// NeuroPLC — Auto-generated IEC 61131-3 SCL
// Graph: kan | Target: S71200Backend
// Work memory: 75KB | LUT points: 15
// Nodes: 11 | Ops: {'matmul': 3, 'standard_act': 2, 'bspline_lut': 2, 'add': 2, 'softmax': 1, 'argmax': 1}


DATA_BLOCK "NeuroPLC_Weights"
{ S7_Optimized_Access := 'FALSE' }
VERSION : 0.1
NON_RETAIN
   STRUCT

   // BsplineLUT 'l0_bspline': grid(15 pts) + table(16×28×15)
   w0 : ARRAY[0..14] OF REAL :=
[-3.0000000, -2.5714286, -2.1428571, -1.7142857, -1.2857143, -0.8571429, -0.4285714, 0.0
    0.4285714, 0.8571429, 1.2857143, 1.7142857, 2.1428571, 2.5714286, 3.0000000];
   w1 : ARRAY[0..6719] OF REAL :=
[-0.0064954, -0.0050089, -0.0033770, -0.0016958, -0.0000479, 0.0014853, 0.0028220, 0.0038805
    0.0045846, 0.0048793, 0.0047147, 0.0040414, 0.0028094, 0.0009775, -0.0013529, -0.0130491
    -0.0087791, -0.0036095, 0.0020238, 0.0073062, 0.0114015, 0.0134733, 0.0126853, 0.0084933
    0.0015210, -0.0073160, -0.0171017, -0.0269205, -0.0358740, -0.0433676, -0.0119517, -0.0074362
    -0.0021026, 0.0035783, 0.0087589, 0.0125698, 0.0141418, 0.0126054, 0.0074143, -0.0006864
    -0.0106286, -0.0213443, -0.0317654, -0.0408502, -0.0480129, -0.0055758, -0.0085337, -0.0109214
    -0.0123673, -0.0124829, -0.0108790, -0.0071661, -0.0009551, 0.0079073, 0.0186290, 0.0301819
    0.0415377, 0.0516683, 0.0595823, 0.0649290, 0.0033017, -0.0018919, -0.0086076, -0.0158108
    -0.0218283, -0.0249507, -0.0234683, -0.0156713, -0.0006975, 0.0189270, 0.0398287, 0.0586340
    0.0719694, 0.0766010, 0.0717208, -0.0145982, -0.0132009, -0.0118636, -0.0105667, -0.0090013
    -0.0068415, -0.0037615, 0.0005645, 0.0063401, 0.0132795, 0.0209750, 0.0290186, 0.0370023
    0.0445224, 0.0512483, 0.0005540, 0.0050713, 0.0109763, 0.0176704, 0.0237023, 0.0275720
    0.0277792, 0.0228238, 0.0116819, -0.0047655, -0.0251609, -0.0481471, -0.0723664, -0.0964808
    -0.1194836, -0.0025839, -0.0029541, -0.0026654, -0.0016455, 0.0000022, 0.0021641, 0.0047267
    0.0075767, 0.0104673, 0.0126194, 0.0131209, 0.0110596, 0.0055231, -0.0043401, -0.0183258
    -0.0085053, -0.0092509, -0.0093235, -0.0085654, -0.0068801, -0.0041745, -0.0003556, 0.0046696
    0.0108291, 0.0173902, 0.0234552, 0.0281264, 0.0305059, 0.0297509, 0.0259743, -0.0022033
    -0.0008497, 0.0003257, 0.0012372, 0.0018995, 0.0023330, 0.0025581, 0.0025952, 0.0024489
    0.0020599, 0.0013534, 0.0002540, -0.0013131, -0.0034131, -0.0059392, 0.0570825, 0.0523418
    0.0441618, 0.0326389, 0.0183960, 0.0020866, -0.0156358, -0.0341180, -0.0527775, -0.0713162
    -0.0895071, -0.1071230, -0.1239369, -0.1396837, -0.1534356, -0.0017276, 0.0135975, 0.0262822
    0.0349414, 0.0388797, 0.0374410, 0.0299697, 0.0158097, -0.0051883, -0.0311484, -0.0596881
    -0.0884251, -0.1149769, -0.1370229, -0.1533197, 0.0417430, 0.0132695, -0.0117596, -0.0313531
    -0.0452569, -0.0533167, -0.0553782, -0.0512872, -0.0412373, -0.0268139, -0.0099504, 0.0074197
    0.0233633, 0.0360149, 0.0446960, 0.0591801, 0.0506987, 0.0420201, 0.0335674, 0.0251025
    0.0163496, 0.0070328, -0.0031239, -0.0142303, -0.0257320, -0.0369083, -0.0470387, -0.0554027
    -0.0613104, -0.0646050, 0.0380552, 0.0305894, 0.0203781, 0.0079362, -0.0053995, -0.0182449
    -0.0292158, -0.0369281, -0.0402260, -0.0388668, -0.0328362, -0.0221198, -0.0067033, 0.0133397
    0.0364058, -0.0794777, -0.0800806, -0.0797186, -0.0782858, -0.0752684, -0.0701291, -0.0623306
    -0.0513354, -0.0369371, -0.0202517, -0.0027264, 0.0141921, 0.0290567, 0.0404752, 0.0480044
    -0.1608721, -0.1544616, -0.1423316, -0.1249372, -0.1034885, -0.0792385, -0.0534405, -0.0273477
    -0.0021188, 0.0214652, 0.0427176, 0.0609519, 0.0754814, 0.0856493, 0.0913159, 0.0539866
    0.0477996, 0.0377296, 0.0240342, 0.0077611, -0.0099963, -0.0281447, -0.0455906, -0.0613476
    -0.0748558, -0.0856624, -0.0933141, -0.0973580, -0.0973787, -0.0936133, 0.0534758, 0.0429142
    0.0305485, 0.0172136, 0.0040506, -0.0077813, -0.0171231, -0.0228160, -0.0239895, -0.0209286
    -0.0142067, -0.0043974, 0.0079257, 0.0221621, 0.0372402, 0.1102775, 0.1072526, 0.1021108
    0.0946131, 0.0838261, 0.0687763, 0.0484902, 0.0219946, -0.0109618, -0.0477404, -0.0849806
    -0.1193216, -0.1474027, -0.1660319, -0.1749534, -0.0983728, -0.0679108, -0.0389890, -0.0138788
    0.0064673, 0.0211730, 0.0293616, 0.0301567, 0.0231331, 0.0096706, -0.0083994, -0.0292456
    -0.0510370, -0.0719598, -0.0905098, -0.1422940, -0.1310264, -0.1130547, -0.0893668, -0.0624104
    -0.0347168, -0.0088174, 0.0127565, 0.0280181, 0.0371596, 0.0409174, 0.0400284, 0.0352292
    0.0272730, 0.0171998, -0.1772897, -0.1588601, -0.1331439, -0.1010212, -0.0656541, -0.0303357
    0.0016410, 0.0269829, 0.0431205, 0.0503784, 0.0498048, 0.0424480, 0.0293561, 0.0116197
    -0.0089316, -0.0924975, -0.0685450, -0.0453334, -0.0240949, -0.0058931, 0.0082184, 0.0171858
    0.0199555, 0.0158568, 0.0057512, -0.0091168, -0.0275026, -0.0481617, -0.0698275, -0.0908472
    -0.0919868, -0.0763941, -0.0599793, -0.0435190, -0.0277131, -0.0132577, -0.0008484, 0.0088188
    0.0152255, 0.0185620, 0.0191960, 0.0174953, 0.0138274, 0.0085720, 0.0023131, -0.1375341
    -0.1143461, -0.0884176, -0.0609049, -0.0337633, -0.0089942, 0.0114009, 0.0254207, 0.0315517
    0.0302322, 0.0223883, 0.0089463, -0.0091677, -0.0309746, -0.0545734, -0.0019394, 0.0037786
    0.0098244, 0.0154883, 0.0197382, 0.0215240, 0.0197951, 0.0135014, 0.0019694, -0.0139657
    -0.0330918, -0.0541969, -0.0760687, -0.0974818, -0.1169787, -0.1755243, -0.1531998, -0.1266178
    -0.0966809, -0.0651036, -0.0336468, -0.0040715, 0.0218613, 0.0427145, 0.0583474, 0.0689429
    0.0746840, 0.0757539, 0.0723667, 0.0652806, -0.0696934, -0.0602897, -0.0487975, -0.0357825
    -0.0218667, -0.0076757, 0.0061653, 0.0190307, 0.0302458, 0.0389377, 0.0441842, 0.0450629
    0.0406516, 0.0301205, 0.0142489, -0.0597138, -0.0559139, -0.0494283, -0.0404261, -0.0294536
    -0.0170791, -0.0038708, 0.0096030, 0.0226738, 0.0342706, 0.0432220, 0.0483568, 0.0485035
    0.0425778, 0.0310126, -0.0605716, -0.0569390, -0.0505317, -0.0415093, -0.0304389, -0.0179108
    -0.0045154, 0.0091569, 0.0224174, 0.0341838, 0.0432753, 0.0485114, 0.0487112, 0.0427819
    0.0311602, -0.0516885, -0.0380645, -0.0247713, -0.0127368, -0.0022508, 0.0064337, 0.0130636
    0.0173857, 0.0192439, 0.0188696, 0.0165911, 0.0127368, 0.0076349, 0.0016172, -0.0049279
    -0.0562407, -0.0516357, -0.0434013, -0.0321080, -0.0191705, -0.0060523, 0.0057832, 0.0148725
    0.0201440, 0.0220925, 0.0216043, 0.0195661, 0.0168642, 0.0143631, 0.0125459, -0.0215669
    -0.0173831, -0.0123562, -0.0067542, -0.0009397, 0.0047195, 0.0098553, 0.0140999, 0.0171329
    0.0188250, 0.0190945, 0.0178597, 0.0150389, 0.0105708, 0.0047481, -0.0566579, -0.0562306
    -0.0548574, -0.0523959, -0.0483627, -0.0422548, -0.0335695, -0.0218037, -0.0067783, 0.0103907
    0.0282635, 0.0454004, 0.0603615, 0.0717702, 0.0793456, -0.0520496, -0.0423928, -0.0325770
    -0.0232095, -0.0144005, -0.0062322, 0.0012138, 0.0078554, 0.0136411, 0.0186406, 0.0229540
    0.0266813, 0.0299225, 0.0327781, 0.0353559, -0.0642884, -0.0507025, -0.0367111, -0.0231770
    -0.0104224, 0.0012616, 0.0115839, 0.0202534, 0.0269396, 0.0311546, 0.0323713, 0.0300626
    0.0237013, 0.0128268, -0.0018600, -0.0367120, -0.0243320, -0.0127388, -0.0027711, 0.0054115
    0.0116887, 0.0159399, 0.0180448, 0.0179132, 0.0155768, 0.0110978, 0.0045382, -0.0040400
    -0.0145496, -0.0264691, -0.1216510, -0.1105591, -0.0941895, -0.0733171, -0.0496326, -0.0248794
    -0.0008011, 0.0208591, 0.0387466, 0.0530622, 0.0643957, 0.0733367, 0.0804749, 0.0863647
    0.0909459, -0.0027857, -0.0084430, -0.0145285, -0.0204270, -0.0250927, -0.0274549, -0.0264427
    -0.0209856, -0.0104698, 0.0038897, 0.0204213, 0.0374528, 0.0533125, 0.0663794, 0.0759185
    0.0129611, 0.0254017, 0.0356314, 0.0425417, 0.0455004, 0.0439032, 0.0371453, 0.0246222
    0.0061932, -0.0164266, -0.0410586, -0.0655236, -0.0876430, -0.1053033, -0.1175339, -0.0247634
    -0.0279660, -0.0288906, -0.0272312, -0.0232430, -0.0172134, -0.0094298, -0.0001796, 0.0101667
    0.0209071, 0.0312566, 0.0404302, 0.0476427, 0.0521333, 0.0535592, -0.1293642, -0.1193707
    -0.1032642, -0.0817289, -0.0568370, -0.0307407, -0.0055918, 0.0164574, 0.0336519, 0.0458234
    0.0532008, 0.0560128, 0.0544880, 0.0488898, 0.0400817, 0.0759348, 0.0751573, 0.0733678
    0.0703268, 0.0651676, 0.0569878, 0.0448845, 0.0279552, 0.0058174, -0.0198302, -0.0467688
    -0.0727795, -0.0956434, -0.1132157, -0.1246400, 0.0752203, 0.0702935, 0.0637723, 0.0558556
    0.0465078, 0.0356797, 0.0233220, 0.0093856, -0.0060020, -0.0220067, -0.0376174, -0.0518232
    -0.0636131, -0.0720135, -0.0767006, -0.1173986, -0.1049409, -0.0871985, -0.0650950, -0.0405694
    -0.0156189, 0.0077592, 0.0275678, 0.0422579, 0.0520735, 0.0577069, 0.0598503, 0.0591959
    0.0564281, 0.0520940, -0.1212512, -0.1127163, -0.0993807, -0.0818294, -0.0613756, -0.0393746
    -0.0171817, 0.0038479, 0.0225291, 0.0383576, 0.0509995, 0.0601208, 0.0653873, 0.0665038
    0.0638503, -0.1056125, -0.1031581, -0.0990820, -0.0934024, -0.0856393, -0.0752838, -0.0618274
    -0.0447613, -0.0239545, -0.0007861, 0.0229867, 0.0456071, 0.0653182, 0.0804434, 0.0907060
    0.0487952, 0.0374115, 0.0242019, 0.0102135, -0.0029327, -0.0135830, -0.0200835, -0.0207803
    -0.0146193, -0.0029447, 0.0122998, 0.0291703, 0.0457231, 0.0600643, 0.0711699, 0.0646500
    0.0612506, 0.0529924, 0.0403731, 0.0250127, 0.0085953, -0.0071945, -0.0206726, -0.0303979
    -0.0359026, -0.0369623, -0.0333526, -0.0248490, -0.0113090, 0.0059815, 0.0825636, 0.0740969
    0.0609729, 0.0435120, 0.0233914, 0.0023661, -0.0178087, -0.0353779, -0.0489058, -0.0582347
    -0.0635260, -0.0649415, -0.0626425, -0.0568210, -0.0481953, 0.0733571, 0.0654811, 0.0543846
    0.0404885, 0.0252671, 0.0102550, -0.0030131, -0.0130025, -0.0185798, -0.0202170, -0.0187870
    -0.0151632, -0.0102187, -0.0048108, 0.0004789, 0.0597846, 0.0506018, 0.0387739, 0.0250072
    0.0108969, -0.0019105, -0.0117689, -0.0170321, -0.0165256, -0.0109636, -0.0015320, 0.0105832
    0.0241959, 0.0381237, 0.0512467, 0.0794086, 0.0712941, 0.0590351, 0.0430848, 0.0252648
    0.0074750, -0.0083842, -0.0204127, -0.0271671, -0.0290304, -0.0268422, -0.0214424, -0.0136706
    -0.0043701, 0.0055541, -0.0189963, -0.0221225, -0.0233823, -0.0223317, -0.0191588, -0.0140878
    -0.0073429, 0.0008515, 0.0102233, 0.0203094, 0.0305988, 0.0405802, 0.0497428, 0.0575804
    0.0636721, 0.0415532, 0.0397687, 0.0360804, 0.0306095, 0.0239207, 0.0166041, 0.0092500
    0.0024485, -0.0033091, -0.0079269, -0.0114082, -0.0137560, -0.0149734, -0.0150717, -0.0142024
    -0.1213656, -0.1098515, -0.0929578, -0.0714629, -0.0470719, -0.0215433, 0.0033646, 0.0258933
    0.0444176, 0.0578437, 0.0652110, 0.0655589, 0.0579266, 0.0414757, 0.0174933, -0.1205001
    -0.1097379, -0.0932614, -0.0718080, -0.0471914, -0.0212873, 0.0040288, 0.0268811, 0.0455475
    0.0589196, 0.0660424, 0.0659608, 0.0577200, 0.0404886, 0.0155879, -0.1202567, -0.1093710
    -0.0927757, -0.0712194, -0.0465306, -0.0206000, 0.0046820, 0.0274247, 0.0458997, 0.0590270
    0.0658889, 0.0655675, 0.0571451, 0.0398251, 0.0149239, -0.0930097, -0.0831860, -0.0703592
    -0.0552040, -0.0386853, -0.0217846, -0.0054833, 0.0092369, 0.0215748, 0.0314497, 0.0389614
    0.0442093, 0.0472932, 0.0483230, 0.0475881, -0.1132518, -0.1079017, -0.0976854, -0.0829627
    -0.0649007, -0.0447129, -0.0236130, -0.0028146, 0.0165543, 0.0337069, 0.0479419, 0.0585582
    0.0648543, 0.0661755, 0.0626742, -0.0815116, -0.0730840, -0.0626569, -0.0507423, -0.0377882
    -0.0242390, -0.0105393, 0.0028667, 0.0155580, 0.0272082, 0.0375145, 0.0461741, 0.0528842
    0.0573621, 0.0596777, -0.1008868, -0.0948195, -0.0856380, -0.0736700, -0.0594149, -0.0433822
    -0.0260816, -0.0080224, 0.0102401, 0.0279682, 0.0443783, 0.0586871, 0.0701108, 0.0779097
    0.0821002, -0.0928198, -0.0838908, -0.0722195, -0.0583813, -0.0431031, -0.0271209, -0.0111703
    0.0040129, 0.0177917, 0.0299241, 0.0402667, 0.0486763, 0.0550096, 0.0591411, 0.0612585
    -0.1192025, -0.1073053, -0.0904778, -0.0695176, -0.0459871, -0.0214926, 0.0023598, 0.0239637
    0.0418163, 0.0548291, 0.0620169, 0.0623945, 0.0549769, 0.0389000, 0.0154086, -0.0679830
    -0.0513064, -0.0341468, -0.0177486, -0.0029976, 0.0092411, 0.0181021, 0.0227202, 0.0224813
    0.0177747, 0.0092409, -0.0024797, -0.0167467, -0.0329079, -0.0501083, -0.1202152, -0.1092289
    -0.0926936, -0.0714178, -0.0472899, -0.0222603, 0.0017207, 0.0227027, 0.0392099, 0.0516649
    0.0609646, 0.0680063, 0.0736871, 0.0788536, 0.0834750, -0.0320415, -0.0206113, -0.0114709
    -0.0052510, -0.0012089, 0.0014771, 0.0036287, 0.0060675, 0.0094544, 0.0138069, 0.0189818
    0.0248359, 0.0312257, 0.0379923, 0.0447006, 0.0660699, 0.0630954, 0.0595871, 0.0554868
    0.0500426, 0.0424626, 0.0319549, 0.0177277, -0.0005979, -0.0217477, -0.0440348, -0.0657718
    -0.0852719, -0.1008953, -0.1118326, 0.0328585, 0.0217698, 0.0119434, 0.0043030, -0.0008504
    -0.0032515, -0.0026349, 0.0012646, 0.0083698, 0.0172324, 0.0260619, 0.0330673, 0.0364579
    0.0345348, 0.0271977, -0.1172725, -0.1090614, -0.0961407, -0.0789738, -0.0588449, -0.0370850
    -0.0150253, 0.0060030, 0.0248866, 0.0413825, 0.0554658, 0.0671113, 0.0762938, 0.0829856
    0.0871120, 0.0788702, 0.0767232, 0.0737037, 0.0696657, 0.0637522, 0.0550650, 0.0427063
    0.0257779, 0.0038922, -0.0212971, -0.0476260, -0.0729304, -0.0950462, -0.1118830, -0.1226330
    0.0424648, 0.0355723, 0.0284807, 0.0217434, 0.0156830, 0.0106090, 0.0068309, 0.0046579
    0.0042683, 0.0053151, 0.0073201, 0.0098052, 0.0122921, 0.0143158, 0.0156396, -0.1141555
    -0.1016998, -0.0839089, -0.0618142, -0.0376349, -0.0136582, 0.0078285, 0.0245378, 0.0347400
    0.0389358, 0.0381833, 0.0335407, 0.0260662, 0.0168141, 0.0067709, -0.1213959, -0.1175703
    -0.1110765, -0.1020365, -0.0903403, -0.0758647, -0.0584862, -0.0380815, -0.0148199, 0.0099586
    0.0346216, 0.0575365, 0.0770708, 0.0916617, 0.1009580, -0.0431900, -0.0438981, -0.0437770
    -0.0425988, -0.0398651, -0.0350619, -0.0276752, -0.0171910, -0.0033860, 0.0128013, 0.0301419
    0.0474065, 0.0633661, 0.0768385, 0.0874577, 0.0019430, -0.0087142, -0.0163489, -0.0201806
    -0.0205530, -0.0178746, -0.0125535, -0.0049983, 0.0043352, 0.0147992, 0.0256987, 0.0363382
    0.0460225, 0.0540709, 0.0600565, 0.0039094, 0.0201128, 0.0296586, 0.0319383, 0.0287980
    0.0222250, 0.0142065, 0.0067297, 0.0014772, -0.0010882, -0.0008081, 0.0024758, 0.0089216
    0.0186273, 0.0306427, 0.0763165, 0.0725086, 0.0658738, 0.0564109, 0.0447281, 0.0314686
    0.0172757, 0.0027923, -0.0114108, -0.0250536, -0.0379287, -0.0498286, -0.0605459, -0.0698632
    -0.0773902, 0.0831831, 0.0795113, 0.0726465, 0.0625293, 0.0497289, 0.0348502, 0.0184983
    0.0012784, -0.0162054, -0.0333528, -0.0495646, -0.0642413, -0.0767837, -0.0866050, -0.0933383
    0.0471839, 0.0355534, 0.0222393, 0.0082356, -0.0048220, -0.0152611, -0.0214091, -0.0215935
    -0.0147504, -0.0022505, 0.0139268, 0.0318021, 0.0493961, 0.0647776, 0.0768565, 0.0713515
    0.0666394, 0.0594218, 0.0498125, 0.0385150, 0.0262667, 0.0138048, 0.0018668, -0.0089300
    -0.0184476, -0.0266677, -0.0335724, -0.0391433, -0.0433604, -0.0461668, -0.0771443, -0.0710582
    -0.0617116, -0.0493296, -0.0350074, -0.0198900, -0.0051224, 0.0081503, 0.0190202, 0.0275273
    0.0339489, 0.0385621, 0.0416443, 0.0434640, 0.0441410, -0.0979009, -0.0862316, -0.0711662
    -0.0531324, -0.0335126, -0.0137440, 0.0047361, 0.0204905, 0.0323993, 0.0406117, 0.0455938
    0.0478122, 0.0477332, 0.0458205, 0.0424930, 0.0944311, 0.0863878, 0.0740996, 0.0580816
    0.0395634, 0.0198158, 0.0001096, -0.0182844, -0.0341089, -0.0461598, -0.0532464, -0.0541781
    -0.0477642, -0.0329385, -0.0108025, 0.0939177, 0.0870638, 0.0758494, 0.0606509, 0.0425458
    0.0226521, 0.0020875, -0.0180299, -0.0364904, -0.0517164, -0.0620384, -0.0657868, -0.0612920
    -0.0470345, -0.0241054, 0.0934611, 0.0864068, 0.0749925, 0.0596162, 0.0413892, 0.0214640
    0.0009928, -0.0188720, -0.0369049, -0.0515887, -0.0613327, -0.0645465, -0.0596398, -0.0451677
    -0.0222238, 0.0570179, 0.0537455, 0.0489764, 0.0428718, 0.0355747, 0.0272273, 0.0179716
    0.0079496, -0.0025564, -0.0127039, -0.0215103, -0.0279928, -0.0311689, -0.0301138, -0.0249110
    0.0460533, 0.0528679, 0.0571354, 0.0582993, 0.0560601, 0.0501329, 0.0402327, 0.0260748
    0.0077565, -0.0130960, -0.0344739, -0.0543687, -0.0707718, -0.0817546, -0.0867803, 0.0621695
    0.0584621, 0.0535885, 0.0476425, 0.0404141, 0.0316758, 0.0212000, 0.0087594, -0.0055780
    -0.0205620, -0.0346468, -0.0462869, -0.0539364, -0.0561275, -0.0527471, 0.0701987, 0.0696979
    0.0675516, 0.0635566, 0.0572396, 0.0481121, 0.0356854, 0.0194707, -0.0006887, -0.0236225
    -0.0478285, -0.0718046, -0.0940486, -0.1131139, -0.1285232, 0.0605322, 0.0579419, 0.0539998
    0.0487406, 0.0420048, 0.0336216, 0.0234203, 0.0112302, -0.0029310, -0.0182922, -0.0338936
    -0.0487758, -0.0619792, -0.0725872, -0.0804313, 0.0925140, 0.0843020, 0.0722705, 0.0569652
    0.0395218, 0.0211099, 0.0028993, -0.0139404, -0.0282564, -0.0389630, -0.0449914, -0.0452728
    -0.0387385, -0.0244341, -0.0033994, 0.0693646, 0.0566685, 0.0426540, 0.0284249, 0.0152002
    0.0042055, -0.0033339, -0.0061924, -0.0035427, 0.0038494, 0.0148200, 0.0282050, 0.0428405
    0.0575849, 0.0716867, 0.0069745, 0.0062506, 0.0064994, 0.0078262, 0.0099654, 0.0126300
    0.0155331, 0.0183876, 0.0208833, 0.0226164, 0.0231599, 0.0220866, 0.0189695, 0.0134287
    0.0059034, 0.0326397, 0.0199406, 0.0098152, 0.0032476, 0.0000372, -0.0000846, 0.0026136
    0.0078633, 0.0152792, 0.0240088, 0.0330832, 0.0415332, 0.0483899, 0.0527224, 0.0542676
    0.0053282, 0.0129482, 0.0183251, 0.0210448, 0.0216541, 0.0207547, 0.0189484, 0.0168371
    0.0149329, 0.0133894, 0.0122708, 0.0116410, 0.0115643, 0.0120930, 0.0130789, -0.0381531
    -0.0262031, -0.0143655, -0.0034747, 0.0060392, 0.0137694, 0.0193090, 0.0222511, 0.0224485
    0.0207927, 0.0184346, 0.0165254, 0.0162159, 0.0186006, 0.0237847, 0.0409369, 0.0423051
    0.0424320, 0.0410951, 0.0380820, 0.0331813, 0.0261813, 0.0168703, 0.0052438, -0.0078751
    -0.0214561, -0.0344691, -0.0458837, -0.0547040, -0.0605266, 0.0091396, 0.0119548, 0.0140948
    0.0154324, 0.0161025, 0.0162550, 0.0160399, 0.0156069, 0.0150929, 0.0145815, 0.0141431
    0.0138481, 0.0137671, 0.0139622, 0.0143534, 0.0721669, 0.0742674, 0.0740355, 0.0712051
    0.0656274, 0.0571602, 0.0456614, 0.0309891, 0.0132578, -0.0063905, -0.0265570, -0.0458430
    -0.0628498, -0.0762186, -0.0852870, -0.0089771, -0.0124859, -0.0142004, -0.0137117, -0.0110339
    -0.0062053, 0.0007355, 0.0097502, 0.0206647, 0.0327626, 0.0451921, 0.0571012, 0.0676379
    0.0759713, 0.0816357, 0.0681135, 0.0717669, 0.0731730, 0.0718734, 0.0674359, 0.0594302
    0.0474258, 0.0309923, 0.0101209, -0.0135104, -0.0378020, -0.0606542, -0.0799673, -0.0937302
    -0.1014727, 0.0066072, 0.0131599, 0.0193168, 0.0245588, 0.0284010, 0.0303603, 0.0299538
    0.0266985, 0.0203090, 0.0112903, 0.0003451, -0.0118241, -0.0245147, -0.0370358, -0.0489014
    -0.1054841, -0.0859640, -0.0655508, -0.0454745, -0.0263027, -0.0085651, 0.0072089, 0.0204895
    0.0308788, 0.0385047, 0.0436267, 0.0465041, 0.0473965, 0.0465646, 0.0442899, 0.0230305
    0.0095048, 0.0011872, -0.0014041, 0.0002786, 0.0046702, 0.0102053, 0.0153185, 0.0186618
    0.0197552, 0.0183360, 0.0141414, 0.0069087, -0.0035626, -0.0163892, -0.1229653, -0.1097450
    -0.0931571, -0.0735213, -0.0519821, -0.0297309, -0.0079594, 0.0121409, 0.0296408, 0.0446615
    0.0575863, 0.0687990, 0.0786830, 0.0875849, 0.0952085, -0.1548740, -0.1414460, -0.1227592
    -0.0991485, -0.0722224, -0.0436623, -0.0151498, 0.0116337, 0.0353166, 0.0557683, 0.0731680
    0.0876950, 0.0995286, 0.1088290, 0.1154228, -0.1086425, -0.0899576, -0.0683922, -0.0451821
    -0.0221343, -0.0010883, 0.0161161, 0.0276392, 0.0321437, 0.0303009, 0.0232844, 0.0122680
    -0.0015748, -0.0170612, -0.0328486, -0.1558141, -0.1408449, -0.1207802, -0.0960685, -0.0684270
    -0.0396461, -0.0115157, 0.0141738, 0.0359979, 0.0539937, 0.0685638, 0.0801109, 0.0890376
    0.0957244, 0.1001640, -0.0616598, -0.0524274, -0.0414076, -0.0290780, -0.0160703, -0.0030250
    0.0094170, 0.0206151, 0.0300767, 0.0379012, 0.0443362, 0.0496289, 0.0540270, 0.0577579
    0.0607039, 0.0925081, 0.0809107, 0.0674662, 0.0525844, 0.0372056, 0.0223005, 0.0088397
    -0.0022058, -0.0100878, -0.0149464, -0.0171444, -0.0170443, -0.0150086, -0.0114080, -0.0067522
    -0.1215551, -0.1098357, -0.0927275, -0.0710164, -0.0464081, -0.0206612, 0.0044657, 0.0272140
    0.0459589, 0.0596108, 0.0672138, 0.0678120, 0.0604495, 0.0442920, 0.0206181, -0.1208857
    -0.1095647, -0.0924934, -0.0704504, -0.0453027, -0.0189797, 0.0065890, 0.0294740, 0.0479249
    0.0609077, 0.0675675, 0.0670493, 0.0584981, 0.0411776, 0.0164150, -0.1205362, -0.1090672
    -0.0918623, -0.0697141, -0.0445053, -0.0181810, 0.0073136, 0.0300334, 0.0482226, 0.0608837
    0.0672086, 0.0663892, 0.0576175, 0.0402015, 0.0154702, -0.0941092, -0.0845557, -0.0718859
    -0.0567428, -0.0400791, -0.0228652, -0.0060714, 0.0093319, 0.0225441, 0.0334438, 0.0420794
    0.0484995, 0.0527524, 0.0548977, 0.0551881, -0.1170871, -0.1116646, -0.1013879, -0.0865732
    -0.0683226, -0.0477831, -0.0261021, -0.0044266, 0.0161521, 0.0347672, 0.0506076, 0.0628627
    0.0707213, 0.0734210, 0.0710410, -0.0823846, -0.0739108, -0.0634201, -0.0514188, -0.0383376
    -0.0246032, -0.0106423, 0.0031187, 0.0162708, 0.0284763, 0.0394149, 0.0487667, 0.0562115
    0.0614492, 0.0645269, -0.0991079, -0.0922577, -0.0822467, -0.0694684, -0.0545329, -0.0380632
    -0.0206821, -0.0030123, 0.0143144, 0.0306304, 0.0452592, 0.0575243, 0.0667490, 0.0722997
    0.0742855, -0.0928475, -0.0838840, -0.0721083, -0.0580921, -0.0425772, -0.0263157, -0.0100593
    0.0054401, 0.0195247, 0.0319125, 0.0424159, 0.0508468, 0.0570176, 0.0607599, 0.0622474
    -0.1203630, -0.1085233, -0.0916387, -0.0704921, -0.0466520, -0.0217322, 0.0026534, 0.0248913
    0.0434635, 0.0572356, 0.0651691, 0.0662254, 0.0593662, 0.0436765, 0.0203970, -0.0680496
    -0.0515522, -0.0344431, -0.0179460, -0.0029658, 0.0096107, 0.0188968, 0.0240060, 0.0243005
    0.0201390, 0.0121289, 0.0008778, -0.0130066, -0.0289036, -0.0459612, -0.1138717, -0.1025615
    -0.0859516, -0.0648777, -0.0412208, -0.0169221, 0.0060774, 0.0258366, 0.0408898, 0.0516737
    0.0591004, 0.0640818, 0.0675302, 0.0703143, 0.0725504, -0.0350313, -0.0229405, -0.0128055
    -0.0053238, 0.0000572, 0.0039619, 0.0070147, 0.0098400, 0.0129439, 0.0163589, 0.0199993
    0.0237792, 0.0276129, 0.0314070, 0.0349383, 0.0761654, 0.0712323, 0.0657907, 0.0599320
    0.0529649, 0.0441535, 0.0327617, 0.0180532, -0.0003224, -0.0211741, -0.0429252, -0.0639990
    -0.0828190, -0.0978532, -0.1083473, 0.0390785, 0.0275469, 0.0171428, 0.0088180, 0.0028944
    -0.0003426, -0.0006074, 0.0023855, 0.0085804, 0.0165564, 0.0245516, 0.0308039, 0.0335512
    0.0311235, 0.0234511, -0.1124076, -0.1048866, -0.0926845, -0.0762174, -0.0567367, -0.0355421
    -0.0139333, 0.0067902, 0.0255361, 0.0420414, 0.0562504, 0.0681074, 0.0775567, 0.0845398
    0.0889506, 0.0777938, 0.0761875, 0.0736788, 0.0700997, 0.0646103, 0.0563323, 0.0443873
    0.0278971, 0.0064857, -0.0182131, -0.0440628, -0.0689272, -0.0906700, -0.1072281, -0.1178123
    0.0306264, 0.0248821, 0.0192516, 0.0142293, 0.0100919, 0.0071031, 0.0055270, 0.0056275
    0.0075227, 0.0107481, 0.0146931, 0.0187473, 0.0223004, 0.0247633, 0.0259229, -0.1100040
    -0.0974996, -0.0798112, -0.0579656, -0.0341471, -0.0106065, 0.0104052, 0.0266372, 0.0363968
    0.0402233, 0.0392138, 0.0344657, 0.0270764, 0.0181347, 0.0085847, -0.1101300, -0.1074096
    -0.1023327, -0.0949400, -0.0850188, -0.0723417, -0.0566813, -0.0378103, -0.0158138, 0.0079732
    0.0319032, 0.0543286, 0.0736020, 0.0881442, 0.0975696, -0.0224207, -0.0236837, -0.0245226
    -0.0247033, -0.0237885, -0.0213294, -0.0168772, -0.0099832, -0.0004217, 0.0111389, 0.0238074
    0.0366923, 0.0489020, 0.0595761, 0.0683924, -0.0233470, -0.0315586, -0.0356521, -0.0350509
    -0.0305355, -0.0229643, -0.0131955, -0.0020877, 0.0095558, 0.0211516, 0.0321712, 0.0420859
    0.0503673, 0.0565039, 0.0602835, -0.0084433, 0.0087051, 0.0199937, 0.0247043, 0.0244047
    0.0207943, 0.0155723, 0.0104381, 0.0068485, 0.0052909, 0.0060104, 0.0092522, 0.0152612
    0.0242227, 0.0352821, 0.0585067, 0.0569909, 0.0533496, 0.0474729, 0.0396850, 0.0303350
    0.0197723, 0.0083458, -0.0035997, -0.0157382, -0.0277479, -0.0393072, -0.0500946, -0.0597806
    -0.0678997, 0.0763782, 0.0748911, 0.0701328, 0.0619394, 0.0508106, 0.0372841, 0.0218974
    0.0051883, -0.0122721, -0.0297793, -0.0465951, -0.0619815, -0.0752003, -0.0855319, -0.0925743
    0.0374300, 0.0266855, 0.0146888, 0.0023938, -0.0087210, -0.0171474, -0.0213768, -0.0199010
    -0.0117905, 0.0015674, 0.0182065, 0.0361603, 0.0534627, 0.0681992, 0.0793608, 0.0584625
    0.0558492, 0.0511390, 0.0443516, 0.0359860, 0.0265690, 0.0166272, 0.0066872, -0.0027968
    -0.0116610, -0.0198142, -0.0271652, -0.0336226, -0.0390905, -0.0433884, -0.0890283, -0.0810995
    -0.0695774, -0.0548310, -0.0381366, -0.0208221, -0.0042159, 0.0103538, 0.0218367, 0.0302932
    0.0360615, 0.0394797, 0.0408862, 0.0406171, 0.0389746, -0.1011540, -0.0898113, -0.0746058
    -0.0559599, -0.0353910, -0.0144791, 0.0051956, 0.0220529, 0.0348570, 0.0437498, 0.0492174
    0.0517461, 0.0518220, 0.0499288, 0.0465025, -0.1150191, -0.1040288, -0.0878393, -0.0671941
    -0.0437533, -0.0192299, 0.0046633, 0.0262135, 0.0438444, 0.0565260, 0.0633650, 0.0634681
    0.0559420, 0.0400093, 0.0169120, -0.1136940, -0.1035435, -0.0878935, -0.0674332, -0.0439016
    -0.0190980, 0.0051784, 0.0271281, 0.0450974, 0.0580147, 0.0649535, 0.0649878, 0.0571912
    0.0407560, 0.0169362, -0.1135426, -0.1032815, -0.0875194, -0.0669554, -0.0433427, -0.0184950
    0.0057740, 0.0276506, 0.0454741, 0.0581963, 0.0649221, 0.0647562, 0.0568036, 0.0402859
    0.0164578, -0.0887678, -0.0792654, -0.0668474, -0.0521640, -0.0361579, -0.0197886, -0.0040159
    0.0102007, 0.0220788, 0.0315445, 0.0387009, 0.0436513, 0.0464988, 0.0473565, 0.0465069
    -0.1083338, -0.1028552, -0.0927300, -0.0783368, -0.0608156, -0.0413501, -0.0211241, -0.0013213
    0.0169684, 0.0330303, 0.0462434, 0.0559867, 0.0616393, 0.0626229, 0.0591023, -0.0775478
    -0.0695332, -0.0595474, -0.0480733, -0.0355557, -0.0224369, -0.0091594, 0.0038346, 0.0161274
    0.0274012, 0.0373626, 0.0457186, 0.0521761, 0.0564617, 0.0586449, -0.0962942, -0.0905587
    -0.0818326, -0.0704136, -0.0567581, -0.0413319, -0.0246004, -0.0070292, 0.0108738, 0.0284328
    0.0449295, 0.0596457, 0.0718633, 0.0809003, 0.0867065, -0.0886533, -0.0800715, -0.0688260
    -0.0554658, -0.0406965, -0.0252327, -0.0097892, 0.0049194, 0.0182786, 0.0300741, 0.0401918
    0.0485174, 0.0549369, 0.0593518, 0.0619392, -0.1129163, -0.1014855, -0.0853049, -0.0651442
    -0.0425303, -0.0190337, 0.0037750, 0.0243255, 0.0411600, 0.0532720, 0.0597679, 0.0597540
    0.0523366, 0.0367359, 0.0141528, -0.0644862, -0.0485097, -0.0320092, -0.0161761, -0.0018866
    0.0100011, 0.0186287, 0.0231381, 0.0229192, 0.0183537, 0.0100715, -0.0012977, -0.0151239
    -0.0307667, -0.0473992, -0.1192922, -0.1084692, -0.0920533, -0.0708351, -0.0467016, -0.0216032
    0.0025099, 0.0236875, 0.0404533, 0.0532275, 0.0629040, 0.0703769, 0.0765402, 0.0822354
    0.0873918, -0.0294734, -0.0189659, -0.0106106, -0.0049696, -0.0013039, 0.0012005, 0.0033573
    0.0059804, 0.0097195, 0.0145674, 0.0203531, 0.0269052, 0.0340527, 0.0416067, 0.0490741
    0.0650349, 0.0627376, 0.0597952, 0.0561095, 0.0509495, 0.0435475, 0.0331361, 0.0189477
    0.0006264, -0.0205367, -0.0428393, -0.0645787, -0.0840523, -0.0996066, -0.1104411, 0.0299549
    0.0195369, 0.0103629, 0.0033123, -0.0013214, -0.0032781, -0.0022979, 0.0018792, 0.0091779
    0.0181812, 0.0271367, 0.0342920, 0.0378948, 0.0362825, 0.0293554, -0.1136357, -0.1055042
    -0.0927660, -0.0758810, -0.0561190, -0.0347965, -0.0132299, 0.0072643, 0.0255859, 0.0414988
    0.0549833, 0.0660195, 0.0745876, 0.0806665, 0.0842130, 0.0796799, 0.0776106, 0.0746405
    0.0706247, 0.0647179, 0.0560345, 0.0436891, 0.0267961, 0.0049771, -0.0201172, -0.0463292
    -0.0715011, -0.0934753, -0.1101679, -0.1207850, 0.0471702, 0.0401892, 0.0328941, 0.0258325
    0.0193094, 0.0136164, 0.0090447, 0.0058856, 0.0043172, 0.0040642, 0.0047380, 0.0059499
    0.0073114, 0.0084452, 0.0091719, -0.1143654, -0.1021862, -0.0845330, -0.0624114, -0.0380585
    -0.0137824, 0.0081091, 0.0253079, 0.0360626, 0.0408471, 0.0406915, 0.0366261, 0.0296812
    0.0208831, 0.0111921, -0.1183035, -0.1140783, -0.1073372, -0.0982326, -0.0866561, -0.0724844
    -0.0555943, -0.0358624, -0.0134468, 0.0103689, 0.0340196, 0.0559402, 0.0745657, 0.0883988
    0.0971212, -0.0449943, -0.0453366, -0.0448266, -0.0432475, -0.0400870, -0.0348164, -0.0269064
    -0.0158281, -0.0013547, 0.0155321, 0.0335481, 0.0514091, 0.0678313, 0.0815803, 0.0922910
    0.0065674, -0.0063583, -0.0157020, -0.0205504, -0.0213812, -0.0187517, -0.0132195, -0.0053419
    0.0043035, 0.0150584, 0.0262445, 0.0371835, 0.0471970, 0.0556191, 0.0620026, 0.0105306
    0.0255404, 0.0339575, 0.0352378, 0.0312270, 0.0239082, 0.0152645, 0.0072789, 0.0016253
    -0.0012590, -0.0012459, 0.0017927, 0.0079849, 0.0174008, 0.0291002, 0.0858274, 0.0804212
    0.0722181, 0.0612891, 0.0482883, 0.0339036, 0.0188229, 0.0037340, -0.0107619, -0.0244099
    -0.0370420, -0.0484899, -0.0585854, -0.0671524, -0.0738745, 0.0880742, 0.0826101, 0.0743533
    0.0633208, 0.0500298, 0.0350263, 0.0188560, 0.0020649, -0.0148010, -0.0311950, -0.0465703
    -0.0603800, -0.0720773, -0.0811279, -0.0872167, 0.0517958, 0.0393813, 0.0254100, 0.0109012
    -0.0025541, -0.0133320, -0.0198087, -0.0203604, -0.0139593, -0.0019614, 0.0136811, 0.0310161
    0.0480916, 0.0630035, 0.0746856, 0.0802013, 0.0737863, 0.0650000, 0.0540316, 0.0416047
    0.0284741, 0.0153943, 0.0031199, -0.0077261, -0.0170466, -0.0248760, -0.0312489, -0.0361996
    -0.0397611, -0.0419380, -0.0813725, -0.0748128, -0.0649224, -0.0519620, -0.0370499, -0.0213537
    -0.0060409, 0.0077209, 0.0190091, 0.0278806, 0.0346374, 0.0395811, 0.0430137, 0.0452262
    0.0463194, -0.0887788, -0.0781593, -0.0643381, -0.0476983, -0.0295392, -0.0112124, 0.0059304
    0.0205375, 0.0315560, 0.0391289, 0.0436976, 0.0457040, 0.0455896, 0.0437931, 0.0406991
    -0.0681019, -0.0558745, -0.0441106, -0.0335166, -0.0238243, -0.0147096, -0.0058486, 0.0030829
    0.0123038, 0.0216121, 0.0307007, 0.0392626, 0.0469907, 0.0535900, 0.0589749, -0.0745009
    -0.0610971, -0.0466884, -0.0322327, -0.0184111, -0.0058885, 0.0046702, 0.0125999, 0.0175007
    0.0200328, 0.0211215, 0.0216920, 0.0226695, 0.0249387, 0.0286753, -0.0721163, -0.0584018
    -0.0438990, -0.0295951, -0.0161466, -0.0041911, 0.0056340, 0.0126911, 0.0166200, 0.0181703
    0.0183687, 0.0182420, 0.0188171, 0.0210736, 0.0251719, -0.0926290, -0.0828816, -0.0707450
    -0.0568312, -0.0417447, -0.0260898, -0.0104708, 0.0045080, 0.0182859, 0.0304758, 0.0407343
    0.0487180, 0.0540833, 0.0565155, 0.0561972, -0.0907978, -0.0859772, -0.0774038, -0.0652007
    -0.0502352, -0.0334171, -0.0156562, 0.0021376, 0.0190963, 0.0345190, 0.0477468, 0.0581205
    0.0649812, 0.0677005, 0.0661841, -0.0552471, -0.0429697, -0.0313496, -0.0211351, -0.0121846
    -0.0043050, 0.0026963, 0.0090124, 0.0147835, 0.0199395, 0.0243578, 0.0279157, 0.0304905
    0.0319690, 0.0324008, -0.0518637, -0.0356115, -0.0191431, -0.0037401, 0.0095546, 0.0197123
    0.0257038, 0.0265003, 0.0214690, 0.0115618, -0.0018731, -0.0174878, -0.0339341, -0.0498954
    -0.0646034, -0.0750934, -0.0627938, -0.0492242, -0.0351928, -0.0212449, -0.0079108, 0.0042793
    0.0147952, 0.0231211, 0.0287994, 0.0313867, 0.0304399, 0.0255157, 0.0162241, 0.0031023
    -0.0756219, -0.0651536, -0.0545072, -0.0442427, -0.0341002, -0.0237729, -0.0129537, -0.0013358
    0.0112176, 0.0241618, 0.0367822, 0.0483640, 0.0581923, 0.0655877, 0.0704843, -0.0199903
    -0.0168361, -0.0138871, -0.0112165, -0.0084661, -0.0052529, -0.0011937, 0.0040943, 0.0108419
    0.0186709, 0.0270508, 0.0354510, 0.0433412, 0.0502094, 0.0558684, -0.0951167, -0.0843383
    -0.0687285, -0.0492257, -0.0279636, -0.0071445, 0.0110293, 0.0243556, 0.0311273, 0.0316189
    0.0266003, 0.0168414, 0.0031120, -0.0137778, -0.0323163, -0.0324504, -0.0335040, -0.0301457
    -0.0224050, -0.0118296, -0.0000543, 0.0112860, 0.0205565, 0.0263758, 0.0283759, 0.0264421
    0.0204599, 0.0103147, -0.0040378, -0.0214172, 0.0946146, 0.0857759, 0.0748829, 0.0623615
    0.0483462, 0.0329548, 0.0163048, -0.0014860, -0.0201712, -0.0389892, -0.0570498, -0.0734627
    -0.0873376, -0.0978102, -0.1044702, 0.0510492, 0.0419094, 0.0334937, 0.0264414, 0.0206468
    0.0159612, 0.0122362, 0.0093230, 0.0070724, 0.0053317, 0.0039475, 0.0027665, 0.0016353
    0.0004161, -0.0007572, -0.1006878, -0.0916718, -0.0785101, -0.0617960, -0.0429373, -0.0233887
    -0.0046048, 0.0119598, 0.0251807, 0.0352542, 0.0427072, 0.0480662, 0.0518579, 0.0545862
    0.0563552, 0.0503459, 0.0532122, 0.0547124, 0.0544169, 0.0517122, 0.0459743, 0.0365792
    0.0229029, 0.0047388, -0.0164501, -0.0387834, -0.0603808, -0.0793618, -0.0939094, -0.1033076
    -0.0408732, -0.0338215, -0.0260637, -0.0179739, -0.0096838, -0.0013109, 0.0070272, 0.0152130
    0.0230338, 0.0298967, 0.0351137, 0.0379967, 0.0378577, 0.0340710, 0.0270941, -0.1021982
    -0.0930440, -0.0790383, -0.0608542, -0.0401324, -0.0185691, 0.0021393, 0.0202965, 0.0346070
    0.0453794, 0.0533228, 0.0591466, 0.0635600, 0.0672356, 0.0702077, 0.0692438, 0.0678171
    0.0636722, 0.0568775, 0.0478867, 0.0371755, 0.0252196, 0.0124947, -0.0004698, -0.0129301
    -0.0240889, -0.0331487, -0.0393122, -0.0418328, -0.0408491, 0.0921181, 0.0916542, 0.0900433
    0.0870802, 0.0819053, 0.0736216, 0.0613323, 0.0441403, 0.0216763, -0.0043176, -0.0315718
    -0.0578167, -0.0807825, -0.0983015, -0.1099787, -0.1119333, -0.1013238, -0.0848411, -0.0631974
    -0.0384422, -0.0127021, 0.0118965, 0.0332272, 0.0495246, 0.0604681, 0.0660983, 0.0664555
    0.0615804, 0.0515728, 0.0375695, -0.0730997, -0.0675506, -0.0572406, -0.0428076, -0.0259146
    -0.0082835, 0.0083640, 0.0223060, 0.0322131, 0.0383257, 0.0412767, 0.0416989, 0.0402252
    0.0374778, 0.0338920, -0.1076191, -0.0973288, -0.0817078, -0.0611327, -0.0375210, -0.0128788
    0.0107878, 0.0314728, 0.0476305, 0.0595576, 0.0680112, 0.0737484, 0.0775264, 0.0800688
    0.0815150, -0.0741057, -0.0625820, -0.0490312, -0.0339187, -0.0182590, -0.0030981, 0.0105180
    0.0215433, 0.0292440, 0.0341347, 0.0370423, 0.0387934, 0.0402149, 0.0420890, 0.0444250
    -0.0928475, -0.0842471, -0.0718093, -0.0558799, -0.0377289, -0.0186795, -0.0000546, 0.0168227
    0.0308220, 0.0415834, 0.0489398, 0.0527240, 0.0527690, 0.0489501, 0.0418835, -0.1074911
    -0.0975065, -0.0823477, -0.0623628, -0.0394076, -0.0154245, 0.0076440, 0.0278558, 0.0436803
    0.0552340, 0.0630454, 0.0676432, 0.0695555, 0.0693021, 0.0672456, -0.1037187, -0.0934545
    -0.0781682, -0.0583332, -0.0359152, -0.0129661, 0.0084626, 0.0263191, 0.0389774, 0.0465126
    0.0494256, 0.0482171, 0.0433880, 0.0354613, 0.0253502, -0.0266544, -0.0336035, -0.0358269
    -0.0331325, -0.0266085, -0.0174167, -0.0067191, 0.0043226, 0.0147216, 0.0241911, 0.0326196
    0.0398955, 0.0459071, 0.0505421, 0.0536739, -0.0570067, -0.0510674, -0.0426060, -0.0319958
    -0.0200086, -0.0074390, 0.0049183, 0.0162687, 0.0258464, 0.0330016, 0.0371130, 0.0375598
    0.0337208, 0.0250448, 0.0121974, -0.0520371, -0.0486492, -0.0428014, -0.0346550, -0.0247561
    -0.0136728, -0.0019731, 0.0097748, 0.0209302, 0.0305615, 0.0376646, 0.0412354, 0.0402695
    0.0338457, 0.0224826, -0.0525712, -0.0493106, -0.0435266, -0.0353693, -0.0253905, -0.0141650
    -0.0022675, 0.0097271, 0.0211668, 0.0310908, 0.0384612, 0.0422399, 0.0413890, 0.0349552
    0.0234615, -0.0436548, -0.0344229, -0.0244913, -0.0145098, -0.0049960, 0.0035400, 0.0105880
    0.0156380, 0.0183099, 0.0187436, 0.0172091, 0.0139763, 0.0093153, 0.0035013, -0.0030965
    -0.0556900, -0.0499911, -0.0410367, -0.0294721, -0.0165975, -0.0037504, 0.0077314, 0.0165105
    0.0216022, 0.0234336, 0.0227849, 0.0204365, 0.0171684, 0.0137455, 0.0106627, -0.0259741
    -0.0219326, -0.0168972, -0.0111316, -0.0050199, 0.0010473, 0.0066791, 0.0114847, 0.0151220
    0.0174439, 0.0183521, 0.0177483, 0.0155340, 0.0116302, 0.0062922, -0.0511092, -0.0508130
    -0.0497722, -0.0478703, -0.0446635, -0.0396890, -0.0324842, -0.0225864, -0.0097885, 0.0050931
    0.0209868, 0.0368205, 0.0515223, 0.0640591, 0.0740691, -0.0455572, -0.0389769, -0.0315846
    -0.0238023, -0.0159021, -0.0081477, -0.0008025, 0.0058698, 0.0116732, 0.0166817, 0.0210367
    0.0248796, 0.0283520, 0.0315941, 0.0347292, -0.0521327, -0.0440120, -0.0343157, -0.0235823
    -0.0124407, -0.0015250, 0.0085306, 0.0170920, 0.0235774, 0.0276143, 0.0288828, 0.0270626
    0.0218338, 0.0129269, 0.0009554, -0.0296755, -0.0206468, -0.0117076, -0.0034971, 0.0036499
    0.0094163, 0.0134849, 0.0155384, 0.0153486, 0.0130434, 0.0088394, 0.0029535, -0.0043976
    -0.0129850, -0.0223708, -0.1298479, -0.1198579, -0.1037237, -0.0821519, -0.0570350, -0.0303334
    -0.0040077, 0.0199815, 0.0400947, 0.0564755, 0.0696887, 0.0802990, 0.0888711, 0.0959336
    0.1013906, -0.0123170, -0.0173108, -0.0223907, -0.0269699, -0.0300543, -0.0306267, -0.0276697
    -0.0201659, -0.0075500, 0.0089352, 0.0275948, 0.0467340, 0.0646579, 0.0797176, 0.0910631
    0.0070675, 0.0216721, 0.0336126, 0.0416478, 0.0452635, 0.0439874, 0.0373472, 0.0248705
    0.0065269, -0.0159460, -0.0403687, -0.0645619, -0.0863460, -0.1036090, -0.1154111, -0.0113047
    -0.0162561, -0.0191668, -0.0195974, -0.0176888, -0.0136153, -0.0075510, 0.0003296, 0.0097397
    0.0199408, 0.0300821, 0.0393124, 0.0467806, 0.0516635, 0.0536200, -0.1079049, -0.0966202
    -0.0809671, -0.0616764, -0.0403355, -0.0185810, 0.0019502, 0.0196217, 0.0331276, 0.0424848
    0.0480414, 0.0501450, 0.0491435, 0.0453990, 0.0395204, 0.0775554, 0.0768969, 0.0750791
    0.0718545, 0.0663915, 0.0578248, 0.0452890, 0.0279188, 0.0053668, -0.0206430, -0.0478687
    -0.0740687, -0.0970009, -0.1144996, -0.1257243, 0.0913561, 0.0854800, 0.0772502, 0.0668551
    0.0543047, 0.0395988, 0.0227372, 0.0037195, -0.0172225, -0.0389295, -0.0600102, -0.0790736
    -0.0947282, -0.1056358, -0.1113782, -0.1320192, -0.1215669, -0.1043566, -0.0811897, -0.0543402
    -0.0261668, 0.0009719, 0.0247173, 0.0431832, 0.0563729, 0.0647624, 0.0688274, 0.0690438
    0.0658983, 0.0600689, -0.1010175, -0.0905779, -0.0776513, -0.0629304, -0.0471000, -0.0308443
    -0.0148477, 0.0002056, 0.0137100, 0.0253749, 0.0349882, 0.0423381, 0.0472127, 0.0494224
    0.0491671, -0.1211558, -0.1172538, -0.1114027, -0.1037132, -0.0937722, -0.0811365, -0.0653627
    -0.0460078, -0.0230143, 0.0021315, 0.0275575, 0.0513916, 0.0717615, 0.0868845, 0.0965336
    0.0494736, 0.0359992, 0.0213548, 0.0067268, -0.0064018, -0.0165311, -0.0221612, -0.0217922
    -0.0144951, -0.0016240, 0.0148963, 0.0331406, 0.0511840, 0.0671452, 0.0799014, 0.0788706
    0.0729088, 0.0622679, 0.0476134, 0.0306091, 0.0129765, -0.0035632, -0.0172888, -0.0267865
    -0.0318731, -0.0326728, -0.0293100, -0.0219089, -0.0106480, 0.0033538, 0.0925338, 0.0821000
    0.0672296, 0.0483524, 0.0271705, 0.0054589, -0.0150071, -0.0324523, -0.0454621, -0.0540636
    -0.0586445, -0.0595926, -0.0572955, -0.0521561, -0.0448425, 0.0690861, 0.0587341, 0.0464455
    0.0326976, 0.0185494, 0.0050934, -0.0065779, -0.0153722, -0.0204912, -0.0223142, -0.0215147
    -0.0187662, -0.0147421, -0.0101061, -0.0053480, 0.0586342, 0.0486394, 0.0362978, 0.0223597
    0.0083873, -0.0040105, -0.0132247, -0.0176466, -0.0161782, -0.0097662, 0.0001318, 0.0120584
    0.0245558, 0.0361959, 0.0460624, 0.0790675, 0.0685686, 0.0549296, 0.0386712, 0.0213098
    0.0044188, -0.0104284, -0.0216584, -0.0280488, -0.0297815, -0.0273896, -0.0214060, -0.0123639
    -0.0008248, 0.0121490, -0.0273778, -0.0298186, -0.0300706, -0.0277089, -0.0230271, -0.0163597
    -0.0080415, 0.0015929, 0.0122118, 0.0234960, 0.0351291, 0.0467950, 0.0581773, 0.0689432
    0.0784699, 0.0476604, 0.0463219, 0.0426467, 0.0367949, 0.0294816, 0.0214537, 0.0134582
    0.0062421, 0.0004070, -0.0040258, -0.0071805, -0.0091812, -0.0101519, -0.0102194, -0.0095578
    0.0304029, 0.0299609, 0.0283810, 0.0258080, 0.0226823, 0.0194614, 0.0166025, 0.0145632
    0.0137208, 0.0141327, 0.0157763, 0.0186291, 0.0226685, 0.0278575, 0.0339104, 0.0345100
    0.0326362, 0.0292712, 0.0247248, 0.0197737, 0.0152209, 0.0118698, 0.0105236, 0.0117567
    0.0152271, 0.0203643, 0.0265975, 0.0333560, 0.0400800, 0.0464014, 0.0338928, 0.0317958
    0.0282599, 0.0236199, 0.0186726, 0.0142415, 0.0111500, 0.0102218, 0.0120325, 0.0161676
    0.0219648, 0.0287619, 0.0358965, 0.0427228, 0.0488790, 0.0046954, 0.0116264, 0.0173569
    0.0214700, 0.0240567, 0.0252368, 0.0251304, 0.0238575, 0.0215543, 0.0184219, 0.0146775
    0.0105383, 0.0062218, 0.0019434, -0.0021083, -0.0191749, -0.0094293, 0.0006520, 0.0101550
    0.0183319, 0.0244443, 0.0277538, 0.0275222, 0.0233902, 0.0165163, 0.0084378, 0.0006922
    -0.0051829, -0.0077142, -0.0065467, 0.0294622, 0.0295048, 0.0293245, 0.0289509, 0.0282756
    0.0271824, 0.0255550, 0.0232769, 0.0202718, 0.0166221, 0.0124502, 0.0078785, 0.0030293
    -0.0019695, -0.0068946, 0.0182424, 0.0192221, 0.0189058, 0.0174219, 0.0154607, 0.0137452
    0.0129981, 0.0139420, 0.0171122, 0.0222932, 0.0290820, 0.0370757, 0.0458710, 0.0550637
    0.0642243, 0.0104603, 0.0148278, 0.0182071, 0.0203796, 0.0215195, 0.0218237, 0.0214891
    0.0207123, 0.0197267, 0.0189108, 0.0186794, 0.0194477, 0.0216304, 0.0256145, 0.0312986
    0.0288828, 0.0303219, 0.0302638, 0.0286950, 0.0260210, 0.0226715, 0.0190761, 0.0156643
    0.0128450, 0.0109435, 0.0102641, 0.0111116, 0.0137901, 0.0185719, 0.0251629, 0.0282172
    0.0247361, 0.0213094, 0.0183155, 0.0160110, 0.0146458, 0.0144697, 0.0157324, 0.0185745
    0.0226995, 0.0277018, 0.0331755, 0.0387150, 0.0439251, 0.0485927, -0.1130037, -0.1031320
    -0.0877097, -0.0674313, -0.0440963, -0.0195678, 0.0042915, 0.0256186, 0.0429744, 0.0566154
    0.0672216, 0.0754733, 0.0820508, 0.0875940, 0.0920447, 0.0132133, 0.0027073, -0.0061052
    -0.0123128, -0.0155831, -0.0156166, -0.0121143, -0.0047768, 0.0064200, 0.0204005, 0.0358140
    0.0513098, 0.0655372, 0.0771829, 0.0855869, 0.0260068, 0.0368160, 0.0451292, 0.0500039
    0.0510243, 0.0478048, 0.0399600, 0.0271043, 0.0092365, -0.0121068, -0.0350051, -0.0575373
    -0.0777829, -0.0938797, -0.1049897, -0.0346115, -0.0298637, -0.0236218, -0.0161368, -0.0078215
    0.0009023, 0.0096125, 0.0178873, 0.0253830, 0.0320698, 0.0379960, 0.0432100, 0.0477603
    0.0516920, 0.0549929, -0.0851682, -0.0732715, -0.0580560, -0.0403095, -0.0214675, -0.0030029
    0.0136117, 0.0269035, 0.0356922, 0.0399670, 0.0400095, 0.0361015, 0.0285244, 0.0176015
    0.0043791, 0.0696061, 0.0698523, 0.0690327, 0.0668753, 0.0626045, 0.0554160, 0.0445053
    0.0290678, 0.0087778, -0.0147759, -0.0395259, -0.0634049, -0.0843453, -0.1003504, -0.1106538
    0.0847614, 0.0817984, 0.0774030, 0.0715933, 0.0639596, 0.0540674, 0.0414825, 0.0257704
    0.0068310, -0.0140993, -0.0354497, -0.0556498, -0.0731287, -0.0863692, -0.0947818, -0.1108918
    -0.1006383, -0.0850245, -0.0647790, -0.0416889, -0.0176021, 0.0056336, 0.0261704, 0.0425557
    0.0549190, 0.0637850, 0.0696785, 0.0731242, 0.0746315, 0.0744391, -0.0359605, -0.0178695
    -0.0014532, 0.0120036, 0.0221845, 0.0288286, 0.0316750, 0.0304629, 0.0251512, 0.0165774
    0.0057988, -0.0061272, -0.0181433, -0.0292130, -0.0386574, -0.0708394, -0.0641480, -0.0559069
    -0.0464048, -0.0356751, -0.0237368, -0.0106088, 0.0036901, 0.0190069, 0.0346515, 0.0497998
    0.0636278, 0.0753113, 0.0840681, 0.0898459, 0.0253482, 0.0136452, 0.0040002, -0.0026618
    -0.0062726, -0.0068129, -0.0042634, 0.0013949, 0.0100250, 0.0208644, 0.0329941, 0.0454952
    0.0574490, 0.0679496, 0.0763194, 0.0761478, 0.0701023, 0.0614798, 0.0506471, 0.0385232
    0.0260594, 0.0142067, 0.0039160, -0.0040498, -0.0096800, -0.0131522, -0.0146441, -0.0143331
    -0.0124082, -0.0092572, 0.0853835, 0.0769114, 0.0653868, 0.0512972, 0.0361628, 0.0215635
    0.0090791, 0.0002895, -0.0036293, -0.0031155, 0.0009886, 0.0078412, 0.0166000, 0.0264176
    0.0363500, 0.0368931, 0.0249396, 0.0148120, 0.0071692, 0.0021551, -0.0001156, 0.0004715
    0.0040309, 0.0105108, 0.0191935, 0.0291949, 0.0396308, 0.0496171, 0.0582856, 0.0650451
    0.0502979, 0.0430935, 0.0364318, 0.0307130, 0.0259937, 0.0223112, 0.0197022, 0.0182039
    0.0177968, 0.0182349, 0.0192161, 0.0204378, 0.0215978, 0.0224020, 0.0226989, 0.0537954
    0.0429471, 0.0322709, 0.0223738, 0.0138986, 0.0074903, 0.0037938, 0.0034542, 0.0068461
    0.0132637, 0.0217306, 0.0312708, 0.0409081, 0.0496822, 0.0569103, -0.0337906, -0.0338268
    -0.0312272, -0.0257847, -0.0181233, -0.0089149, 0.0011688, 0.0114562, 0.0213738, 0.0307424
    0.0394810, 0.0475086, 0.0547444, 0.0610953, 0.0662584, 0.0881414, 0.0805324, 0.0699557
    0.0567018, 0.0419037, 0.0267425, 0.0123994, 0.0000555, -0.0093472, -0.0158243, -0.0196306
    -0.0210208, -0.0202498, -0.0175845, -0.0135008, -0.0354648, -0.0236547, -0.0141773, -0.0076552
    -0.0032492, -0.0000366, 0.0029056, 0.0065003, 0.0114475, 0.0175556, 0.0244101, 0.0315964
    0.0387001, 0.0453171, 0.0512239, -0.0439950, -0.0284136, -0.0145570, -0.0034529, 0.0050194
    0.0110466, 0.0148154, 0.0165123, 0.0164307, 0.0152895, 0.0139141, 0.0131302, 0.0137632
    0.0165923, 0.0215903, -0.0426016, -0.0268748, -0.0129865, -0.0019827, 0.0062605, 0.0119343
    0.0152297, 0.0163380, 0.0155698, 0.0137140, 0.0116790, 0.0103730, 0.0107044, 0.0135302
    0.0188134, -0.0765257, -0.0629248, -0.0492052, -0.0360816, -0.0233384, -0.0107067, 0.0020828
    0.0152990, 0.0290268, 0.0426143, 0.0552256, 0.0660244, 0.0741749, 0.0788853, 0.0801361
    -0.0903997, -0.0838859, -0.0738837, -0.0605716, -0.0447450, -0.0272350, -0.0088723, 0.0095121
    0.0270972, 0.0431015, 0.0567535, 0.0672814, 0.0739139, 0.0759257, 0.0734005, -0.0290878
    -0.0193884, -0.0107825, -0.0037935, 0.0019271, 0.0067775, 0.0111563, 0.0154618, 0.0199955
    0.0246714, 0.0293064, 0.0337173, 0.0377211, 0.0411402, 0.0438918, -0.0324730, -0.0145571
    0.0022114, 0.0164322, 0.0272931, 0.0340158, 0.0358218, 0.0319329, 0.0219057, 0.0066369
    -0.0126418, -0.0346985, -0.0583015, -0.0822319, -0.1054924, -0.0558906, -0.0409747, -0.0268090
    -0.0142774, -0.0032717, 0.0063735, 0.0148234, 0.0222434, 0.0286298, 0.0333042, 0.0354189
    0.0341266, 0.0285796, 0.0179952, 0.0027153, -0.0409851, -0.0315624, -0.0236506, -0.0176629
    -0.0127711, -0.0080759, -0.0026780, 0.0043219, 0.0135128, 0.0242417, 0.0355454, 0.0464605
    0.0560237, 0.0633141, 0.0681491, 0.0050864, 0.0031617, 0.0012772, -0.0002720, -0.0010702
    -0.0006945, 0.0012780, 0.0052700, 0.0115048, 0.0194068, 0.0282008, 0.0371117, 0.0453642
    0.0522132, 0.0574377, -0.0753358, -0.0628220, -0.0470761, -0.0290922, -0.0105453, 0.0068506
    0.0213813, 0.0313329, 0.0353606, 0.0335961, 0.0265405, 0.0146951, -0.0014392, -0.0212990
    -0.0432361, -0.0184157, -0.0207121, -0.0186254, -0.0120949, -0.0026898, 0.0079273, 0.0180935
    0.0261462, 0.0306967, 0.0314534, 0.0283988, 0.0215154, 0.0107857, -0.0037451, -0.0209390
    0.1098743, 0.0971976, 0.0831130, 0.0683380, 0.0529351, 0.0369295, 0.0203462, 0.0032103
    -0.0143455, -0.0317586, -0.0483590, -0.0634763, -0.0764404, -0.0865966, -0.0935558, 0.0509910
    0.0430018, 0.0359005, 0.0302400, 0.0257608, 0.0221569, 0.0191224, 0.0163511, 0.0136112
    0.0109670, 0.0085569, 0.0065195, 0.0049932, 0.0041148, 0.0039949, -0.0854806, -0.0765071
    -0.0641224, -0.0488998, -0.0320135, -0.0146719, 0.0019160, 0.0165418, 0.0282655, 0.0372225
    0.0438169, 0.0484528, 0.0515343, 0.0534496, 0.0543095, 0.0467085, 0.0500092, 0.0519840
    0.0521990, 0.0500837, 0.0450599, 0.0365493, 0.0239738, 0.0071411, -0.0125975, -0.0335047
    -0.0538431, -0.0718754, -0.0859206, -0.0952787, -0.0230177, -0.0165606, -0.0097636, -0.0030205
    0.0034271, 0.0093464, 0.0145047, 0.0186690, 0.0216335, 0.0232993, 0.0235941, 0.0224459
    0.0197827, 0.0155572, 0.0101577, -0.0921038, -0.0821922, -0.0683197, -0.0511887, -0.0321903
    -0.0127554, 0.0056855, 0.0217016, 0.0342108, 0.0435254, 0.0503060, 0.0552137, 0.0589091
    0.0620186, 0.0645688, 0.0845091, 0.0829789, 0.0785135, 0.0711270, 0.0610952, 0.0487090
    0.0342591, 0.0180363, 0.0004978, -0.0172333, -0.0338675, -0.0481154, -0.0586876, -0.0643650
    -0.0651538, 0.1137435, 0.1152690, 0.1146520, 0.1115171, 0.1049914, 0.0941736, 0.0781623
    0.0560562, 0.0275396, -0.0053602, -0.0400299, -0.0738565, -0.1042268, -0.1286379, -0.1465044
    -0.1684104, -0.1501535, -0.1249484, -0.0940938, -0.0602001, -0.0259531, 0.0059613, 0.0328573
    0.0525943, 0.0652115, 0.0712935, 0.0714247, 0.0661896, 0.0562088, 0.0427307, -0.0503977
    -0.0506114, -0.0448492, -0.0333775, -0.0181797, -0.0013379, 0.0150659, 0.0289498, 0.0386589
    0.0442467, 0.0461941, 0.0449820, 0.0410910, 0.0350124, 0.0274207, -0.1653357, -0.1475474
    -0.1235737, -0.0940846, -0.0614347, -0.0280754, 0.0035420, 0.0309662, 0.0523038, 0.0678938
    0.0786333, 0.0854193, 0.0891490, 0.0906904, 0.0904086, -0.1087819, -0.0884275, -0.0671555
    -0.0457646, -0.0251207, -0.0060936, 0.0104469, 0.0236312, 0.0328709, 0.0387032, 0.0419465
    0.0434195, 0.0439407, 0.0442931, 0.0446437, -0.1266607, -0.1110010, -0.0915719, -0.0691153
    -0.0450837, -0.0209704, 0.0017312, 0.0215279, 0.0371565, 0.0482746, 0.0547700, 0.0565305
    0.0534438, 0.0454575, 0.0335584, -0.1570769, -0.1387548, -0.1151947, -0.0871013, -0.0566182
    -0.0259717, 0.0026120, 0.0269067, 0.0451943, 0.0577899, 0.0655168, 0.0691983, 0.0696577
    0.0677052, 0.0639231, -0.1261191, -0.1114090, -0.0917283, -0.0678558, -0.0419078, -0.0160775
    0.0074419, 0.0264572, 0.0392942, 0.0463550, 0.0485604, 0.0468315, 0.0420893, 0.0352507
    0.0271612, 0.0016886, -0.0034076, -0.0062224, -0.0065271, -0.0046582, -0.0009845, 0.0041250
    0.0103016, 0.0171778, 0.0243929, 0.0315875, 0.0384022, 0.0444778, 0.0494593, 0.0530685
    -0.0586066, -0.0488042, -0.0374860, -0.0252883, -0.0128322, -0.0007379, 0.0103744, 0.0198843
    0.0271202, 0.0312048, 0.0312092, 0.0262046, 0.0152623, -0.0024403, -0.0258767, -0.0726769
    -0.0606264, -0.0462496, -0.0304846, -0.0146020, 0.0001086, 0.0123575, 0.0208551, 0.0245597
    0.0234212, 0.0176375, 0.0074066, -0.0070738, -0.0255599, -0.0470098, -0.0701338, -0.0576829
    -0.0431355, -0.0274767, -0.0119804, 0.0020633, 0.0133642, 0.0206320, 0.0228561, 0.0201438
    0.0128822, 0.0014583, -0.0137410, -0.0322948, -0.0531948, -0.0279673, -0.0286247, -0.0272538
    -0.0237653, -0.0185474, -0.0120157, -0.0045860, 0.0033262, 0.0113115, 0.0189863, 0.0259732
    0.0318948, 0.0363739, 0.0390544, 0.0399516, -0.0148245, -0.0203611, -0.0253312, -0.0289826
    -0.0306585, -0.0297070, -0.0254767, -0.0173158, -0.0050234, 0.0098001, 0.0251034, 0.0388354
    0.0489449, 0.0534696, 0.0519917, -0.0399748, -0.0329524, -0.0258572, -0.0190899, -0.0126072
    -0.0063407, -0.0002217, 0.0058184, 0.0118013, 0.0175614, 0.0228865, 0.0275640, 0.0313816
    0.0341366, 0.0357966, -0.0285481, -0.0222452, -0.0142416, -0.0050878, 0.0041539, 0.0123920
    0.0185347, 0.0214906, 0.0204473, 0.0157097, 0.0078617, -0.0025123, -0.0148284, -0.0284944
    -0.0427786, -0.0257903, -0.0232106, -0.0191659, -0.0138036, -0.0075587, -0.0008831, 0.0057715
    0.0119532, 0.0172025, 0.0210281, 0.0229308, 0.0224117, 0.0189716, 0.0121562, 0.0022918
    -0.0556407, -0.0492407, -0.0405992, -0.0300930, -0.0183685, -0.0060876, 0.0060879, 0.0174960
    0.0273625, 0.0344634, 0.0374622, 0.0350226, 0.0258082, 0.0086118, -0.0155212, -0.0246833
    -0.0134096, -0.0030787, 0.0054715, 0.0119456, 0.0160791, 0.0176076, 0.0162670, 0.0118661
    0.0045076, -0.0056325, -0.0183781, -0.0335533, -0.0509503, -0.0698107, 0.0758282, 0.0712990
    0.0637114, 0.0532410, 0.0403873, 0.0256688, 0.0096038, -0.0072893, -0.0244861, -0.0414381
    -0.0575904, -0.0723883, -0.0852773, -0.0957080, -0.1032286, -0.0272636, -0.0054069, 0.0130674
    0.0265102, 0.0347065, 0.0375231, 0.0348273, 0.0264861, 0.0126950, -0.0050363, -0.0248699
    -0.0449679, -0.0634921, -0.0786596, -0.0896422, 0.0212463, 0.0060381, -0.0068306, -0.0162102
    -0.0219605, -0.0239996, -0.0222455, -0.0166161, -0.0072543, 0.0047986, 0.0182762, 0.0319124
    0.0444409, 0.0546325, 0.0619014, 0.0601048, 0.0539238, 0.0468514, 0.0392553, 0.0312255
    0.0228358, 0.0141603, 0.0052728, -0.0037557, -0.0128655, -0.0219997, -0.0311016, -0.0401143
    -0.0489769, -0.0575546, 0.0505073, 0.0433356, 0.0343323, 0.0240723, 0.0136213, 0.0040730
    -0.0034789, -0.0079406, -0.0085177, -0.0056126, 0.0000731, 0.0078375, 0.0169790, 0.0267895
    0.0364471, -0.0636398, -0.0618810, -0.0584648, -0.0534031, -0.0466455, -0.0381379, -0.0278261
    -0.0156560, -0.0017405, 0.0131396, 0.0280368, 0.0420032, 0.0540911, 0.0633837, 0.0694982
    -0.1056871, -0.1005495, -0.0924400, -0.0816240, -0.0684469, -0.0532590, -0.0364103, -0.0182510
    0.0007787, 0.0198783, 0.0381573, 0.0547250, 0.0686909, 0.0791922, 0.0858493, 0.0747247
    0.0698360, 0.0618605, 0.0510159, 0.0378837, 0.0230666, 0.0071670, -0.0092124, -0.0254645
    -0.0409627, -0.0550762, -0.0671738, -0.0766244, -0.0828237, -0.0856321, 0.0446811, 0.0333259
    0.0211552, 0.0091630, -0.0015313, -0.0098010, -0.0145196, -0.0145603, -0.0092444, 0.0003156
    0.0125592, 0.0259260, 0.0388556, 0.0498322, 0.0581175, 0.0824134, 0.0793522, 0.0751757
    0.0698541, 0.0627653, 0.0532534, 0.0406626, 0.0243368, 0.0040534, -0.0186773, -0.0419116
    -0.0637060, -0.0821168, -0.0952939, -0.1030124, -0.0624190, -0.0492911, -0.0344611, -0.0190550
    -0.0044665, 0.0078954, 0.0166216, 0.0203030, 0.0179868, 0.0105443, -0.0006970, -0.0144097
    -0.0292662, -0.0439499, -0.0573317, -0.1098224, -0.0966860, -0.0796248, -0.0593739, -0.0375329
    -0.0157511, 0.0043221, 0.0210374, 0.0331596, 0.0411098, 0.0457233, 0.0478353, 0.0482811
    0.0478677, 0.0469099, -0.1029273, -0.0934337, -0.0783636, -0.0582396, -0.0353691, -0.0121622
    0.0089709, 0.0256202, 0.0358804, 0.0398652, 0.0381929, 0.0314821, 0.0203511, 0.0054623
    -0.0117558, -0.0129940, 0.0032964, 0.0167624, 0.0264253, 0.0319798, 0.0331593, 0.0296970
    0.0213262, 0.0080899, -0.0087311, -0.0275466, -0.0467662, -0.0647995, -0.0800937, -0.0917489
    -0.0516169, -0.0437829, -0.0348672, -0.0252163, -0.0152860, -0.0055387, 0.0035635, 0.0115582
    0.0180818, 0.0231653, 0.0269382, 0.0295301, 0.0310706, 0.0316869, 0.0314655, -0.0606097
    -0.0479242, -0.0336796, -0.0186602, -0.0043078, 0.0078987, 0.0164799, 0.0199566, 0.0173295
    0.0095186, -0.0020760, -0.0160546, -0.0310172, -0.0455792, -0.0586256, -0.0023447, 0.0054930
    0.0125585, 0.0180971, 0.0216683, 0.0228493, 0.0212176, 0.0163508, 0.0080439, -0.0030367
    -0.0160067, -0.0299821, -0.0440787, -0.0574138, -0.0691312, -0.1130826, -0.1027315, -0.0871549
    -0.0667522, -0.0434779, -0.0193757, 0.0035107, 0.0231375, 0.0378977, 0.0479302, 0.0538104
    0.0561138, 0.0554160, 0.0522932, 0.0473337, 0.0261008, 0.0237962, 0.0210699, 0.0181847
    0.0154457, 0.0131608, 0.0116376, 0.0111837, 0.0120514, 0.0142701, 0.0178137, 0.0226561
    0.0287710, 0.0361154, 0.0443497, 0.0389122, 0.0331583, 0.0262795, 0.0188822, 0.0118818
    0.0062118, 0.0028056, 0.0025965, 0.0062087, 0.0130295, 0.0221370, 0.0326092, 0.0435241
    0.0539819, 0.0634644, 0.0371999, 0.0310599, 0.0239560, 0.0165273, 0.0096815, 0.0043420
    0.0014320, 0.0018750, 0.0062709, 0.0139274, 0.0238286, 0.0349590, 0.0463029, 0.0568719
    0.0661554, 0.0063919, 0.0157115, 0.0229632, 0.0275294, 0.0295813, 0.0293358, 0.0270096
    0.0228194, 0.0170354, 0.0101414, 0.0026749, -0.0048270, -0.0118269, -0.0178046, -0.0225394
    -0.0176481, -0.0088305, 0.0010414, 0.0109957, 0.0198356, 0.0263512, 0.0293328, 0.0275704
    0.0204287, 0.0095694, -0.0027713, -0.0143571, -0.0229518, -0.0264136, -0.0242404, 0.0393840
    0.0371946, 0.0349346, 0.0327545, 0.0304749, 0.0278979, 0.0248253, 0.0210592, 0.0164724
    0.0112225, 0.0055381, -0.0003522, -0.0062199, -0.0118377, -0.0170046, 0.0184495, 0.0151031
    0.0100581, 0.0037712, -0.0025648, -0.0077151, -0.0104446, -0.0095185, -0.0041011, 0.0050465
    0.0167636, 0.0298897, 0.0432643, 0.0557583, 0.0667895, 0.0112919, 0.0156397, 0.0185222
    0.0197031, 0.0194920, 0.0182298, 0.0162573, 0.0139155, 0.0115625, 0.0096260, 0.0085512
    0.0087831, 0.0107669, 0.0149163, 0.0211033, 0.0234623, 0.0254973, 0.0260349, 0.0249826
    0.0226724, 0.0194610, 0.0157049, 0.0117606, 0.0080322, 0.0051139, 0.0036475, 0.0042747
    0.0076371, 0.0143209, 0.0239440, 0.0187196, 0.0155459, 0.0127765, 0.0107508, 0.0096177
    0.0095150, 0.0105808, 0.0129528, 0.0167047, 0.0216524, 0.0275477, 0.0341422, 0.0411875
    0.0484340, 0.0556083, -0.1306002, -0.1193450, -0.1021170, -0.0796934, -0.0539429, -0.0267968
    -0.0001862, 0.0239575, 0.0441187, 0.0604437, 0.0734940, 0.0838316, 0.0920182, 0.0985813
    0.1034534, 0.0107884, -0.0053214, -0.0192264, -0.0296043, -0.0358746, -0.0374991, -0.0339398
    -0.0246584, -0.0095535, 0.0097296, 0.0311092, 0.0525034, 0.0718304, 0.0870774, 0.0974331
    0.0031126, 0.0206697, 0.0351923, 0.0452271, 0.0502242, 0.0496853, 0.0431122, 0.0300067
    0.0103543, -0.0139243, -0.0404249, -0.0667432, -0.0904748, -0.1092905, -0.1221657, -0.0520697
    -0.0468236, -0.0397836, -0.0312404, -0.0216104, -0.0113175, -0.0007852, 0.0095626, 0.0193661
    0.0285202, 0.0369838, 0.0447156, 0.0516744, 0.0578191, 0.0631074, -0.1170136, -0.1049505
    -0.0873950, -0.0652318, -0.0406834, -0.0160495, 0.0063705, 0.0242772, 0.0358551, 0.0412259
    0.0409956, 0.0357699, 0.0261548, 0.0127960, -0.0029647, 0.0778834, 0.0782785, 0.0774099
    0.0749514, 0.0700255, 0.0617234, 0.0491357, 0.0313535, 0.0080131, -0.0190674, -0.0475246
    -0.0749948, -0.0991146, -0.1176003, -0.1295576, 0.0977556, 0.0937919, 0.0877881, 0.0798047
    0.0695575, 0.0567425, 0.0410558, 0.0221934, 0.0001788, -0.0236541, -0.0476441, -0.0701296
    -0.0894495, -0.1039978, -0.1131355, -0.1318879, -0.1202315, -0.1023184, -0.0789717, -0.0522220
    -0.0241692, 0.0030867, 0.0274456, 0.0472358, 0.0624983, 0.0737025, 0.0813174, 0.0858125
    0.0876475, 0.0871170, -0.0787815, -0.0625625, -0.0442741, -0.0251577, -0.0066410, 0.0098378
    0.0228404, 0.0309285, 0.0330955, 0.0300616, 0.0229786, 0.0129985, 0.0012730, -0.0110558
    -0.0230188, -0.1118863, -0.1068451, -0.0997779, -0.0908730, -0.0799020, -0.0666127, -0.0507528
    -0.0320701, -0.0106198, 0.0123119, 0.0351317, 0.0562457, 0.0740605, 0.0870611, 0.0951032
    0.0519505, 0.0387175, 0.0242196, 0.0096593, -0.0034003, -0.0133752, -0.0186815, -0.0177354
    -0.0095692, 0.0043197, 0.0218175, 0.0408104, 0.0591847, 0.0748816, 0.0868012, 0.0919732
    0.0815943, 0.0675893, 0.0505740, 0.0319630, 0.0132169, -0.0042040, -0.0188390, -0.0295005
    -0.0360906, -0.0387846, -0.0377573, -0.0331837, -0.0252767, -0.0149074, 0.0922140, 0.0813033
    0.0655480, 0.0455295, 0.0234068, 0.0014300, -0.0181512, -0.0330867, -0.0415979, -0.0437899
    -0.0402392, -0.0315222, -0.0182153, -0.0009476, 0.0187303, 0.0536413, 0.0412279, 0.0280402
    0.0148872, 0.0030660, -0.0060982, -0.0112801, -0.0111547, -0.0048893, 0.0063776, 0.0210151
    0.0373921, 0.0538775, 0.0688694, 0.0812733, 0.0584316, 0.0504765, 0.0413359, 0.0314795
    0.0216659, 0.0126701, 0.0052672, 0.0002324, -0.0018778, -0.0013814, 0.0011853, 0.0052857
    0.0103835, 0.0159422, 0.0214276, 0.0783539, 0.0672679, 0.0529166, 0.0360236, 0.0185715
    0.0026148, -0.0097917, -0.0165932, -0.0163414, -0.0100139, 0.0008054, 0.0145327, 0.0295838
    0.0443949, 0.0577488, -0.0106321, -0.0160237, -0.0194384, -0.0202431, -0.0184938, -0.0142861
    -0.0077158, 0.0011216, 0.0120269, 0.0243861, 0.0374821, 0.0505972, 0.0630142, 0.0740194
    0.0829627, 0.1128316, 0.1014200, 0.0860184, 0.0670208, 0.0459345, 0.0243306, 0.0037801
    -0.0141457, -0.0281803, -0.0382758, -0.0446886, -0.0476752, -0.0474922, -0.0444139, -0.0390233
    -0.0816246, -0.0697223, -0.0568112, -0.0435949, -0.0302681, -0.0169962, -0.0039447, 0.0087209
    0.0207962, 0.0319213, 0.0416975, 0.0497259, 0.0556077, 0.0589738, 0.0599692, -0.0879650
    -0.0758476, -0.0611801, -0.0448164, -0.0277903, -0.0111458, 0.0040730, 0.0168220, 0.0263104
    0.0327600, 0.0366460, 0.0384434, 0.0386274, 0.0376709, 0.0360120, -0.0859623, -0.0735822
    -0.0588253, -0.0425716, -0.0258403, -0.0096586, 0.0049464, 0.0169475, 0.0255829, 0.0311529
    0.0342235, 0.0353603, 0.0351293, 0.0340890, 0.0326688, -0.0966872, -0.0865728, -0.0736831
    -0.0586674, -0.0422918, -0.0253293, -0.0085529, 0.0072645, 0.0214393, 0.0336460, 0.0436484
    0.0512103, 0.0560956, 0.0580938, 0.0574425, -0.0945337, -0.0894433, -0.0802962, -0.0672610
    -0.0513152, -0.0334823, -0.0147862, 0.0037494, 0.0211786, 0.0368669, 0.0502576, 0.0607939
    0.0679192, 0.0711006, 0.0702231, -0.0619982, -0.0498987, -0.0378336, -0.0265377, -0.0160327
    -0.0062993, 0.0026818, 0.0109300, 0.0184325, 0.0250491, 0.0306077, 0.0349360, 0.0378619
    0.0392279, 0.0391305, -0.0656302, -0.0510966, -0.0352784, -0.0192829, -0.0042040, 0.0088649
    0.0188305, 0.0245995, 0.0254002, 0.0217478, 0.0144789, 0.0044302, -0.0075615, -0.0206643
    -0.0341306, -0.0826330, -0.0706524, -0.0567626, -0.0417494, -0.0263137, -0.0111514, 0.0030415
    0.0155690, 0.0257838, 0.0332323, 0.0375096, 0.0382110, 0.0349314, 0.0273172, 0.0159059
    -0.0859155, -0.0748173, -0.0625717, -0.0498051, -0.0366276, -0.0231194, -0.0093609, 0.0045676
    0.0184861, 0.0318155, 0.0438772, 0.0539924, 0.0614825, 0.0657124, 0.0668081, -0.0346492
    -0.0263255, -0.0186206, -0.0119624, -0.0060421, -0.0005087, 0.0049890, 0.0108019, 0.0171526
    0.0237505, 0.0301762, 0.0360104, 0.0408340, 0.0442495, 0.0462393, -0.1087883, -0.0976977
    -0.0809710, -0.0595461, -0.0357161, -0.0118519, 0.0096756, 0.0264956, 0.0367549, 0.0406727
    0.0389855, 0.0324303, 0.0217438, 0.0076968, -0.0083495, -0.0314350, -0.0309183, -0.0269287
    -0.0195517, -0.0099757, 0.0005476, 0.0107664, 0.0194289, 0.0254537, 0.0284416, 0.0281640
    0.0243921, 0.0168972, 0.0055154, -0.0087866, 0.0910923, 0.0843453, 0.0755951, 0.0650978
    0.0528062, 0.0386553, 0.0225804, 0.0045166, -0.0153938, -0.0361809, -0.0566676, -0.0756769
    -0.0920318, -0.1045899, -0.1128105, 0.0450460, 0.0364813, 0.0286870, 0.0223081, 0.0173337
    0.0137155, 0.0114050, 0.0103536, 0.0104454, 0.0112943, 0.0124466, 0.0134486, 0.0138468
    0.0132154, 0.0116173, -0.1108743, -0.1016423, -0.0876293, -0.0694293, -0.0486008, -0.0267581
    -0.0055155, 0.0135128, 0.0290574, 0.0412281, 0.0504796, 0.0572665, 0.0620434, 0.0652467
    0.0669944, 0.0627705, 0.0644517, 0.0647949, 0.0634283, 0.0596446, 0.0527171, 0.0419192
    0.0265243, 0.0062714, -0.0172378, -0.0419358, -0.0657552, -0.0866286, -0.1025591, -0.1127767
    -0.0218376, -0.0169390, -0.0115866, -0.0060391, -0.0004291, 0.0051179, 0.0104764, 0.0155210
    0.0200745, 0.0237526, 0.0261195, 0.0267391, 0.0251756, 0.0210380, 0.0147203, -0.1099808
    -0.0996387, -0.0839987, -0.0638262, -0.0409644, -0.0173183, 0.0052071, 0.0247069, 0.0397294
    0.0506370, 0.0582455, 0.0633709, 0.0668289, 0.0693983, 0.0712120, 0.0294770, 0.0320434
    0.0324159, 0.0304823, 0.0267890, 0.0219203, 0.0164603, 0.0109933, 0.0060412, 0.0018761
    -0.0012920, -0.0032532, -0.0037977, -0.0027394, -0.0003045, 0.0717664, 0.0720363, 0.0713655
    0.0695558, 0.0659256, 0.0597655, 0.0503660, 0.0370179, 0.0194285, -0.0010284, -0.0225621
    -0.0433819, -0.0616971, -0.0757966, -0.0853504, -0.0971435, -0.0888121, -0.0751265, -0.0566303
    -0.0350977, -0.0123739, 0.0096960, 0.0292672, 0.0447979, 0.0559610, 0.0627324, 0.0650884
    0.0630051, 0.0565055, 0.0464294, -0.0590174, -0.0519605, -0.0419014, -0.0294713, -0.0157986
    -0.0020402, 0.0106469, 0.0211055, 0.0284799, 0.0331183, 0.0356704, 0.0367856, 0.0371135
    0.0372755, 0.0374068, -0.0827147, -0.0742662, -0.0615940, -0.0450193, -0.0260955, -0.0064469
    0.0123021, 0.0285274, 0.0409846, 0.0499503, 0.0560810, 0.0600333, 0.0624638, 0.0640005
    0.0647741, -0.0470894, -0.0367588, -0.0256586, -0.0142252, -0.0030874, 0.0071149, 0.0157418
    0.0221536, 0.0259360, 0.0275773, 0.0277913, 0.0272920, 0.0267931, 0.0269720, 0.0278670
    -0.0727474, -0.0668466, -0.0578925, -0.0460417, -0.0321625, -0.0171638, -0.0019545, 0.0125563
    0.0255665, 0.0367001, 0.0456880, 0.0522612, 0.0561505, 0.0571126, 0.0553561, -0.0863063
    -0.0783605, -0.0660394, -0.0496105, -0.0306195, -0.0106859, 0.0085710, 0.0255317, 0.0389144
    0.0487864, 0.0555529, 0.0596186, 0.0613887, 0.0612618, 0.0595291, -0.0949871, -0.0859515
    -0.0720920, -0.0538049, -0.0329108, -0.0113116, 0.0090905, 0.0263934, 0.0390809, 0.0471812
    0.0511082, 0.0512762, 0.0480991, 0.0420099, 0.0337679, -0.0401284, -0.0424569, -0.0406399
    -0.0346944, -0.0256664, -0.0146609, -0.0027832, 0.0088618, 0.0193528, 0.0285045, 0.0363158
    0.0427852, 0.0479114, 0.0516898, 0.0540555, -0.1809668, -0.1611378, -0.1350816, -0.1040773
    -0.0700176, -0.0348307, -0.0004444, 0.0312131, 0.0582302, 0.0787604, 0.0909738, 0.0930401
    0.0831294, 0.0596091, 0.0242863, -0.1893306, -0.1691384, -0.1418755, -0.1089427, -0.0727127
    -0.0356141, -0.0000754, 0.0314747, 0.0567998, 0.0744306, 0.0830901, 0.0815010, 0.0683861
    0.0426436, 0.0062217, -0.1878797, -0.1673510, -0.1398640, -0.1068516, -0.0706976, -0.0338406
    0.0012810, 0.0322288, 0.0567745, 0.0735308, 0.0813203, 0.0789659, 0.0652905, 0.0392863
    0.0028980, -0.1256921, -0.1109178, -0.0930693, -0.0731224, -0.0520200, -0.0307028, -0.0101116
    0.0088128, 0.0252721, 0.0390384, 0.0500265, 0.0581510, 0.0633266, 0.0654900, 0.0649650
    -0.1489690, -0.1461080, -0.1358327, -0.1182012, -0.0946844, -0.0668340, -0.0362018, -0.0043397
    0.0271680, 0.0566078, 0.0822336, 0.1022994, 0.1150590, 0.1188704, 0.1138995, -0.1066970
    -0.0934832, -0.0786536, -0.0629892, -0.0467533, -0.0301793, -0.0135005, 0.0030496, 0.0191838
    0.0343995, 0.0481402, 0.0598496, 0.0689712, 0.0749812, 0.0779230, -0.1348043, -0.1243794
    -0.1103693, -0.0934113, -0.0741922, -0.0534015, -0.0317288, -0.0098639, 0.0114574, 0.0313132
    0.0487353, 0.0627554, 0.0724052, 0.0767842, 0.0761707, -0.1243821, -0.1102836, -0.0934975
    -0.0749117, -0.0551993, -0.0350210, -0.0150374, 0.0040909, 0.0217389, 0.0374249, 0.0507028
    0.0611268, 0.0682507, 0.0716656, 0.0716087, -0.1738079, -0.1546682, -0.1298207, -0.1004401
    -0.0681157, -0.0344608, -0.0010886, 0.0303876, 0.0582546, 0.0803986, 0.0946058, 0.0986621
    0.0903540, 0.0676826, 0.0323968, -0.0974979, -0.0732573, -0.0490690, -0.0266834, -0.0069859
    0.0091876, 0.0210012, 0.0276190, 0.0284089, 0.0235534, 0.0134387, -0.0015491, -0.0210238
    -0.0445533, -0.0709084, -0.1071494, -0.0937777, -0.0762404, -0.0555160, -0.0332489, -0.0111220
    0.0091816, 0.0259792, 0.0380258, 0.0458275, 0.0503284, 0.0524727, 0.0532043, 0.0534295
    0.0533965, -0.0464890, -0.0283236, -0.0134692, -0.0030370, 0.0037540, 0.0077936, 0.0099717
    0.0111782, 0.0121589, 0.0130846, 0.0139820, 0.0148780, 0.0157992, 0.0167677, 0.0177216
    0.0817749, 0.0736548, 0.0657425, 0.0583326, 0.0505852, 0.0415955, 0.0304584, 0.0162690
    -0.0014840, -0.0217377, -0.0430355, -0.0639210, -0.0829376, -0.0986629, -0.1102684, 0.0697012
    0.0494400, 0.0314295, 0.0171846, 0.0068191, 0.0003664, -0.0021399, -0.0006664, 0.0045078
    0.0118545, 0.0195327, 0.0257016, 0.0285204, 0.0262353, 0.0186082, -0.1404537, -0.1332769
    -0.1198258, -0.1004744, -0.0767890, -0.0504043, -0.0229552, 0.0039235, 0.0288582, 0.0515203
    0.0718420, 0.0897559, 0.1051943, 0.1180707, 0.1279673, 0.0740729, 0.0726753, 0.0705312
    0.0674477, 0.0625226, 0.0548130, 0.0433757, 0.0272679, 0.0060567, -0.0186492, -0.0447308
    -0.0700692, -0.0925455, -0.1101082, -0.1218789, 0.0116962, 0.0068679, 0.0022397, -0.0016906
    -0.0044297, -0.0054845, -0.0043620, -0.0005691, 0.0061483, 0.0150875, 0.0253068, 0.0358646
    0.0458192, 0.0542469, 0.0605370, -0.0980225, -0.0826218, -0.0635821, -0.0421253, -0.0201336
    0.0004730, 0.0177745, 0.0298510, 0.0353158, 0.0349154, 0.0299298, 0.0216390, 0.0113230
    0.0002465, -0.0105874, -0.1231156, -0.1240876, -0.1211544, -0.1140556, -0.1027111, -0.0870508
    -0.0670047, -0.0425028, -0.0138317, 0.0172964, 0.0488126, 0.0786481, 0.1047340, 0.1250765
    0.1389871, -0.0145934, -0.0187642, -0.0224967, -0.0254090, -0.0270613, -0.0270103, -0.0248126
    -0.0200250, -0.0124217, -0.0026474, 0.0084357, 0.0199655, 0.0310796, 0.0409447, 0.0492299
    -0.0103032, -0.0155723, -0.0187426, -0.0193605, -0.0175851, -0.0136108, -0.0076318, 0.0001577
    0.0094535, 0.0195113, 0.0294770, 0.0384965, 0.0457156, 0.0503173, 0.0521324, -0.0224093
    -0.0045062, 0.0077755, 0.0137654, 0.0149545, 0.0129579, 0.0093906, 0.0058677, 0.0038138
    0.0038912, 0.0065716, 0.0123268, 0.0216286, 0.0348612, 0.0508849, 0.0424644, 0.0422852
    0.0403149, 0.0363429, 0.0304703, 0.0228156, 0.0134979, 0.0026359, -0.0096167, -0.0229660
    -0.0370833, -0.0516399, -0.0663070, -0.0807267, -0.0940333, 0.0839102, 0.0858832, 0.0827519
    0.0741201, 0.0607856, 0.0436144, 0.0234729, 0.0012274, -0.0222692, -0.0462157, -0.0698244
    -0.0923074, -0.1128767, -0.1307397, -0.1450197, 0.0311719, 0.0213974, 0.0097797, -0.0026916
    -0.0141454, -0.0226595, -0.0263122, -0.0231815, -0.0120632, 0.0053756, 0.0267502, 0.0496756
    0.0717670, 0.0906997, 0.1051930, 0.0540827, 0.0536278, 0.0503560, 0.0441418, 0.0355394
    0.0251420, 0.0135425, 0.0013342, -0.0109375, -0.0229174, -0.0342982, -0.0447722, -0.0540322
    -0.0617698, -0.0676644, -0.0724230, -0.0666327, -0.0573684, -0.0448530, -0.0303051, -0.0150007
    -0.0002158, 0.0127737, 0.0229501, 0.0303286, 0.0351824, 0.0377850, 0.0384098, 0.0373328
    0.0348772, -0.1361503, -0.1166962, -0.0937136, -0.0678653, -0.0407226, -0.0139094, 0.0109504
    0.0322331, 0.0486550, 0.0602932, 0.0675648, 0.0708870, 0.0706771, 0.0673626, 0.0615537
    -0.0544687, -0.0437051, -0.0339206, -0.0257257, -0.0186905, -0.0123257, -0.0061415, 0.0003516
    0.0075280, 0.0153015, 0.0234708, 0.0318345, 0.0401914, 0.0483395, 0.0560684, -0.0608231
    -0.0484472, -0.0357842, -0.0237200, -0.0127125, -0.0031949, 0.0043998, 0.0096381, 0.0123318
    0.0132714, 0.0134921, 0.0140293, 0.0159184, 0.0201393, 0.0267115, -0.0586514, -0.0459981
    -0.0332560, -0.0213379, -0.0106801, -0.0016912, 0.0052200, 0.0096447, 0.0114312, 0.0114556
    0.0108510, 0.0107506, 0.0122875, 0.0165336, 0.0234917, -0.0858279, -0.0771211, -0.0662417
    -0.0537299, -0.0400997, -0.0258639, -0.0115350, 0.0023744, 0.0153772, 0.0270885, 0.0371491
    0.0451995, 0.0508804, 0.0538591, 0.0542661, -0.0830688, -0.0783669, -0.0703665, -0.0591938
    -0.0456123, -0.0304227, -0.0144253, 0.0015793, 0.0168279, 0.0307055, 0.0426343, 0.0520366
    0.0583344, 0.0609765, 0.0598729, -0.0502365, -0.0390050, -0.0285038, -0.0194173, -0.0115685
    -0.0047308, 0.0013222, 0.0068169, 0.0119253, 0.0166008, 0.0207425, 0.0242492, 0.0270199
    0.0289598, 0.0300837, -0.0446438, -0.0291118, -0.0136525, 0.0004917, 0.0123509, 0.0209703
    0.0253955, 0.0246719, 0.0182426, 0.0071423, -0.0071967, -0.0233421, -0.0398616, -0.0553618
    -0.0691287, -0.0685240, -0.0572247, -0.0448541, -0.0321555, -0.0195998, -0.0076418, 0.0032634
    0.0126608, 0.0201016, 0.0251612, 0.0274213, 0.0264636, 0.0218697, 0.0132700, 0.0011454
    -0.0622465, -0.0534327, -0.0448424, -0.0369279, -0.0292993, -0.0215185, -0.0131471, -0.0037469
    0.0069450, 0.0184893, 0.0302713, 0.0416763, 0.0520897, 0.0609206, 0.0679912, -0.0116632
    -0.0111671, -0.0106619, -0.0100445, -0.0089517, -0.0070055, -0.0038279, 0.0009593, 0.0075815
    0.0156539, 0.0246390, 0.0339994, 0.0431977, 0.0517109, 0.0592670, -0.0881229, -0.0781274
    -0.0636395, -0.0455383, -0.0258273, -0.0065740, 0.0101536, 0.0222878, 0.0282235, 0.0282068
    0.0229467, 0.0131520, -0.0004683, -0.0171637, -0.0354557, -0.0310612, -0.0332037, -0.0307646
    -0.0237087, -0.0136109, -0.0021387, 0.0090404, 0.0182591, 0.0241067, 0.0261997, 0.0244114
    0.0186152, 0.0086845, -0.0054370, -0.0225773, 0.0912010, 0.0825108, 0.0717202, 0.0592607
    0.0453386, 0.0301472, 0.0138796, -0.0032708, -0.0210114, -0.0386523, -0.0554042, -0.0704778
    -0.0830836, -0.0924566, -0.0982498, 0.0445877, 0.0366656, 0.0293876, 0.0232948, 0.0182583
    0.0141104, 0.0106836, 0.0078105, 0.0053462, 0.0032369, 0.0014513, -0.0000417, -0.0012732
    -0.0022647, -0.0028660, -0.0916373, -0.0829665, -0.0706754, -0.0553336, -0.0382025, -0.0205837
    -0.0037783, 0.0109121, 0.0224901, 0.0311731, 0.0374821, 0.0419384, 0.0450631, 0.0473544
    0.0489128, 0.0457431, 0.0486750, 0.0502555, 0.0500690, 0.0475725, 0.0422156, 0.0334481
    0.0207198, 0.0038610, -0.0157745, -0.0364523, -0.0564381, -0.0739975, -0.0874542, -0.0961460
    -0.0413939, -0.0341401, -0.0262699, -0.0181942, -0.0100675, -0.0020297, 0.0057794, 0.0132201
    0.0200821, 0.0258742, 0.0300352, 0.0320034, 0.0312175, 0.0271721, 0.0203366, -0.0967057
    -0.0885844, -0.0758250, -0.0590212, -0.0396950, -0.0194222, 0.0002216, 0.0176610, 0.0316848
    0.0425407, 0.0508410, 0.0571978, 0.0622234, 0.0664958, 0.0699977, 0.0751898, 0.0734925
    0.0688727, 0.0613898, 0.0514813, 0.0396063, 0.0262238, 0.0117930, -0.0031421, -0.0176976
    -0.0309048, -0.0417947, -0.0493986, -0.0528062, -0.0521251, 0.0895937, 0.0894340, 0.0880990
    0.0853568, 0.0803499, 0.0721848, 0.0599678, 0.0428055, 0.0203328, -0.0057020, -0.0330220
    -0.0593503, -0.0824102, -0.1000266, -0.1117994, -0.1096518, -0.0991899, -0.0830117, -0.0618419
    -0.0376858, -0.0126219, 0.0112708, 0.0319136, 0.0475809, 0.0579588, 0.0630867, 0.0630037
    0.0577492, 0.0474226, 0.0331748, -0.0719742, -0.0677083, -0.0583675, -0.0445441, -0.0279792
    -0.0104798, 0.0061468, 0.0200935, 0.0299511, 0.0359021, 0.0385269, 0.0384058, 0.0361193
    0.0322452, 0.0273153, -0.1082191, -0.0984045, -0.0832039, -0.0629709, -0.0396055, -0.0150965
    0.0085671, 0.0293966, 0.0458561, 0.0582221, 0.0672242, 0.0735919, 0.0780547, 0.0813078
    0.0834462, -0.0804086, -0.0698078, -0.0566190, -0.0412569, -0.0248436, -0.0085425, 0.0064836
    0.0190715, 0.0283846, 0.0348923, 0.0393903, 0.0426747, 0.0455410, 0.0487393, 0.0522195
    -0.0932103, -0.0845391, -0.0719569, -0.0558387, -0.0375244, -0.0184094, 0.0001108, 0.0166410
    0.0299986, 0.0398537, 0.0460892, 0.0485880, 0.0472331, 0.0419531, 0.0334698, -0.1085612
    -0.0991084, -0.0843581, -0.0646322, -0.0417892, -0.0177758, 0.0054612, 0.0259751, 0.0422268
    0.0543071, 0.0627147, 0.0679479, 0.0705053, 0.0708762, 0.0693885, -0.1003418, -0.0904174
    -0.0756939, -0.0566330, -0.0351154, -0.0131038, 0.0074396, 0.0245524, 0.0366783, 0.0438858
    0.0466498, 0.0454450, 0.0407460, 0.0330500, 0.0232421, -0.0159199, -0.0251207, -0.0296165
    -0.0291185, -0.0246507, -0.0173125, -0.0082033, 0.0015776, 0.0110866, 0.0200033, 0.0281632
    0.0354017, 0.0415543, 0.0464564, 0.0499434, 0.1041947, 0.0958120, 0.0828091, 0.0656970
    0.0457254, 0.0241864, 0.0023720, -0.0184257, -0.0368583, -0.0513511, -0.0602730, -0.0619931
    -0.0548803, -0.0374612, -0.0110067, 0.1031948, 0.0958750, 0.0837872, 0.0673266, 0.0476460
    0.0259418, 0.0034103, -0.0187521, -0.0392135, -0.0561000, -0.0674021, -0.0711104, -0.0652155
    -0.0478865, -0.0204032, 0.1026869, 0.0951488, 0.0828476, 0.0662011, 0.0463966, 0.0246650
    0.0022375, -0.0196547, -0.0396644, -0.0559807, -0.0666764, -0.0698245, -0.0634979, -0.0459437
    -0.0184425, 0.0615510, 0.0579486, 0.0527094, 0.0460376, 0.0381558, 0.0292873, 0.0196556
    0.0094842, -0.0008810, -0.0106050, -0.0187300, -0.0242985, -0.0263530, -0.0239989, -0.0174398
    0.0586204, 0.0638330, 0.0666092, 0.0664333, 0.0628905, 0.0555719, 0.0440685, 0.0279712
    0.0073203, -0.0160473, -0.0398455, -0.0617881, -0.0795890, -0.0910551, -0.0956105, 0.0671970
    0.0632501, 0.0580307, 0.0516681, 0.0440047, 0.0348668, 0.0240806, 0.0114723, -0.0028425
    -0.0175906, -0.0312095, -0.0421364, -0.0488089, -0.0497488, -0.0449499, 0.0760260, 0.0755233
    0.0731757, 0.0687844, 0.0619107, 0.0521018, 0.0389052, 0.0218683, 0.0008965, -0.0226720
    -0.0471407, -0.0708135, -0.0919939, -0.1090566, -0.1216133, 0.0652230, 0.0624144, 0.0581192
    0.0524043, 0.0451713, 0.0363124, 0.0257197, 0.0132856, -0.0009080, -0.0160192, -0.0310165
    -0.0448684, -0.0565430, -0.0650609, -0.0703480, 0.1025495, 0.0941380, 0.0815089, 0.0651902
    0.0463273, 0.0261006, 0.0056907, -0.0137219, -0.0308950, -0.0443406, -0.0525089, -0.0538504
    -0.0468153, -0.0300040, -0.0046258, 0.0787182, 0.0650277, 0.0499006, 0.0345391, 0.0202537
    0.0083612, 0.0001782, -0.0029784, -0.0002032, 0.0077642, 0.0197729, 0.0346721, 0.0513109
    0.0685536, 0.0855287, 0.0204548, 0.0188118, 0.0175636, 0.0168812, 0.0166653, 0.0168014
    0.0171746, 0.0176704, 0.0181197, 0.0181358, 0.0172781, 0.0151056, 0.0111775, 0.0051003
    -0.0026946, 0.0419706, 0.0269564, 0.0151480, 0.0076841, 0.0041825, 0.0041738, 0.0071885
    0.0127570, 0.0203212, 0.0289682, 0.0376963, 0.0455041, 0.0513898, 0.0543967, 0.0543478
    -0.0066461, 0.0032795, 0.0108349, 0.0154818, 0.0178441, 0.0186123, 0.0184771, 0.0181289
    0.0181352, 0.0185713, 0.0193894, 0.0205416, 0.0219800, 0.0236485, 0.0253465, -0.0370001
    -0.0231177, -0.0097403, 0.0021514, 0.0121109, 0.0197225, 0.0245706, 0.0262395, 0.0246294
    0.0209045, 0.0165449, 0.0130308, 0.0118423, 0.0143849, 0.0207651, 0.0495908, 0.0504240
    0.0498653, 0.0477044, 0.0437130, 0.0376624, 0.0293235, 0.0184673, 0.0050908, -0.0099062
    -0.0253977, -0.0402578, -0.0533609, -0.0636164, -0.0705508, -0.0032044, 0.0004078, 0.0035714
    0.0061272, 0.0082299, 0.0100522, 0.0117669, 0.0135467, 0.0155198, 0.0176357, 0.0197992
    0.0219152, 0.0238886, 0.0256219, 0.0269743, 0.0804896, 0.0845488, 0.0854426, 0.0828194
    0.0767513, 0.0673350, 0.0546673, 0.0388448, 0.0201683, -0.0002449, -0.0210736, -0.0409962
    -0.0586914, -0.0728720, -0.0828461, 0.0061883, 0.0017653, -0.0016791, -0.0035894, -0.0035622
    -0.0012033, 0.0038817, 0.0120873, 0.0235391, 0.0372878, 0.0521156, 0.0668044, 0.0801363
    0.0909227, 0.0984879, 0.0782531, 0.0823873, 0.0841013, 0.0828612, 0.0780886, 0.0692025
    0.0556220, 0.0367661, 0.0125601, -0.0150451, -0.0435922, -0.0706241, -0.0936836, -0.1104135
    -0.1201997, 0.0117500, 0.0188515, 0.0255360, 0.0312256, 0.0353167, 0.0372044, 0.0362838
    0.0319498, 0.0238475, 0.0126227, -0.0008292, -0.0156123, -0.0308310, -0.0456077, -0.0593798
    -0.0873712, -0.0684245, -0.0491887, -0.0308394, -0.0138055, 0.0015270, 0.0147724, 0.0255446
    0.0335681, 0.0390081, 0.0421403, 0.0432401, 0.0425831, 0.0404468, 0.0371410, 0.0307153
    0.0133339, 0.0024117, -0.0013546, 0.0002400, 0.0052572, 0.0117588, 0.0178065, 0.0217400
    0.0230110, 0.0213489, 0.0164834, 0.0081440, -0.0038699, -0.0185418, -0.1128260, -0.1024632
    -0.0881151, -0.0699771, -0.0492891, -0.0273512, -0.0054634, 0.0150743, 0.0332486, 0.0491932
    0.0633282, 0.0760742, 0.0878514, 0.0990316, 0.1091408, -0.1528460, -0.1425121, -0.1257175
    -0.1026594, -0.0751820, -0.0452239, -0.0147237, 0.0143799, 0.0404992, 0.0634506, 0.0834012
    0.1005182, 0.1149691, 0.1268936, 0.1359573, -0.1018433, -0.0836372, -0.0623418, -0.0392276
    -0.0162838, 0.0044594, 0.0209717, 0.0312229, 0.0337579, 0.0294225, 0.0196379, 0.0058250
    -0.0105951, -0.0281989, -0.0455241, -0.1493881, -0.1373549, -0.1192862, -0.0955012, -0.0678888
    -0.0384277, -0.0090970, 0.0181244, 0.0416509, 0.0614694, 0.0779600, 0.0915027, 0.1024778
    0.1112367, 0.1176324, -0.0349331, -0.0279529, -0.0197789, -0.0107610, -0.0013090, 0.0081634
    0.0172427, 0.0255154, 0.0326687, 0.0387933, 0.0440807, 0.0487222, 0.0529093, 0.0568115
    0.0602173, 0.1205544, 0.1058188, 0.0887534, 0.0698828, 0.0503392, 0.0312895, 0.0139010
    -0.0006595, -0.0114822, -0.0186872, -0.0226522, -0.0237545, -0.0223717, -0.0188926, -0.0138998];

   // MatMul 'l0_base': W(16×28) + b(16)
   w2 : ARRAY[0..463] OF REAL :=
[-0.0013882, -0.0441315, -0.0497092, 0.0728803, 0.1172757, 0.0557204, -0.1279281, -0.0140936
    0.0275907, -0.0084342, -0.1333183, -0.1616967, 0.0622880, -0.0594389, 0.0043229, 0.0611738
    0.1220259, -0.1058920, 0.0347188, -0.1740287, -0.0860635, 0.0561647, 0.0253270, -0.1559720
    -0.0001806, -0.0593703, -0.1082066, 0.1408983, 0.0082371, 0.0615350, 0.0606271, -0.0139833
    0.0006025, 0.0000052, 0.1024181, 0.0426312, -0.0368083, -0.0692211, 0.1015044, 0.0978756
    -0.1267395, 0.0786163, 0.0795663, -0.1321867, -0.0837473, 0.0727976, 0.0891497, 0.1075353
    0.1029092, -0.0491616, -0.0962761, 0.0036916, 0.0764521, 0.0012560, 0.0870020, -0.0370219
    0.0057886, 0.0594535, 0.0492539, 0.0599910, 0.0991477, 0.0759784, 0.1034839, 0.0765070
    -0.0064536, -0.1154565, 0.0978961, 0.0537450, -0.1233592, 0.0735522, 0.1053082, -0.1308326
    0.0207383, 0.0060595, 0.1201932, 0.1152718, 0.0842907, 0.0000465, -0.1089887, -0.1191539
    0.1062245, -0.0721070, 0.0740447, 0.0670456, 0.0433771, -0.0171170, -0.0047695, -0.0493451
    -0.1219756, -0.0765940, -0.1317902, -0.0917500, 0.0516161, 0.1209587, 0.0252934, 0.0791543
    0.0051135, 0.0024225, -0.0783374, 0.0095173, -0.1233951, 0.1139544, -0.1127663, -0.0750138
    0.0528974, 0.0072524, 0.1176932, 0.1416898, -0.0544584, 0.1253684, 0.0776663, -0.0283814
    0.0137591, 0.0569388, 0.0453289, 0.0677023, 0.1082360, 0.0799180, 0.0938548, 0.0771544
    0.0069746, -0.1108984, 0.0846730, 0.0416950, -0.1188783, 0.0658088, 0.1057792, -0.1265364
    0.0360418, 0.0045785, 0.1153241, 0.0904170, 0.0865469, 0.0087526, -0.0958778, -0.1192973
    0.1090868, -0.0666362, 0.0696053, 0.0722429, 0.0056462, 0.0586356, 0.0490777, 0.0578361
    0.0923828, 0.0736616, 0.1067788, 0.0759070, -0.0069964, -0.1113202, 0.1014701, 0.0590277
    -0.1222657, 0.0745245, 0.1014469, -0.1292026, 0.0104095, 0.0133595, 0.1148991, 0.1216200
    0.0856750, -0.0019447, -0.1064186, -0.1109978, 0.1019267, -0.0679926, 0.0763431, 0.0623527
    0.0836457, 0.0294823, 0.0227684, 0.0783483, 0.1014587, 0.0410230, -0.1059015, 0.0075200
    0.0944678, 0.0805901, -0.0332031, -0.0283769, -0.1108075, -0.0058579, 0.0724348, -0.1093511
    0.0532184, 0.0831195, -0.0667785, -0.1254009, 0.0879736, 0.0521980, 0.1006085, 0.0411577
    0.0823388, 0.0909907, 0.0590997, 0.0791134, 0.0062052, 0.0789691, 0.0812276, -0.0065828
    0.0046604, 0.0068373, 0.0909732, 0.0388490, -0.0393353, -0.0595769, 0.1198951, 0.1269972
    -0.1306157, 0.0846802, 0.0600682, -0.1352401, -0.1394826, 0.1113394, 0.0590963, 0.1146857
    0.1164338, -0.0398067, -0.0706691, -0.0047837, 0.0682722, -0.0023853, 0.1131011, -0.0310528
    0.0512412, 0.0684077, 0.0711208, -0.0214811, -0.0435925, -0.0302585, 0.1054738, 0.0198779
    0.0388856, 0.0637241, 0.1051288, 0.1087856, -0.1198317, 0.0658411, 0.0124578, -0.1190893
    -0.1069564, 0.0926895, -0.0639997, 0.1092676, 0.0961708, -0.0447814, 0.0403531, 0.0828495
    0.0263916, 0.0700621, 0.0820600, -0.0457664, 0.0803593, 0.0274887, 0.0239213, 0.1015691
    0.1059202, 0.0427109, -0.1471568, 0.0034694, 0.0995782, 0.0763367, -0.0240944, -0.0152521
    -0.0994511, -0.0061452, 0.0722495, -0.1035513, 0.0092637, 0.0696368, -0.0853209, -0.1850126
    0.0793389, 0.0519782, 0.1186866, 0.0409093, 0.0858331, 0.0814064, 0.0419918, 0.0840153
    -0.0649314, -0.0953428, -0.1023471, 0.0550378, 0.0965156, 0.0466747, -0.0809210, 0.0080256
    -0.0215680, -0.1336389, -0.1117073, -0.1125575, 0.0788464, -0.0643976, 0.0481159, 0.0842268
    0.1026619, -0.1040474, 0.0832301, -0.1090984, -0.0836866, 0.0579396, 0.0040390, -0.1291443
    0.0450454, -0.0917196, -0.0974251, 0.0789141, 0.0684333, 0.0900734, 0.0931177, -0.0432523
    -0.0724658, -0.0352811, 0.0934245, 0.0181812, 0.0312624, 0.0841460, 0.1170927, 0.1251855
    -0.1352594, 0.0751825, 0.0115898, -0.1388265, -0.1239149, 0.1147220, -0.0462421, 0.1098945
    0.1214973, -0.0560798, -0.0074267, 0.1178625, 0.0233631, 0.0823163, 0.1092210, -0.0834540
    0.0832089, 0.0483249, 0.0403908, 0.0782055, 0.1009623, 0.0501602, -0.0707420, 0.0286006
    0.0892998, 0.0622746, 0.0043924, -0.0084739, -0.1225706, 0.0187156, 0.0871333, -0.1204818
    0.0278716, 0.0855064, -0.0114739, -0.0986967, 0.0909739, 0.0409267, 0.0783337, 0.0116696
    0.0871308, 0.0808635, 0.0683307, 0.0760468, 0.0281681, 0.0594189, 0.0464249, 0.0876040
    0.1982936, 0.1070388, 0.0929669, 0.0948840, 0.0206189, -0.1665370, 0.0563233, 0.0167750
    -0.1176801, 0.0557749, 0.1595425, -0.1309439, 0.0674684, -0.0237252, 0.1681987, 0.0617818
    0.0804414, 0.0176113, -0.1151736, -0.2100232, 0.1609497, -0.1076512, 0.0576393, 0.1076324
    0.0815907, 0.0256319, 0.0198486, 0.0768283, 0.0914778, 0.0391061, -0.1091738, 0.0041704
    0.0922172, 0.0892048, -0.0379398, -0.0292676, -0.1045256, -0.0106281, 0.0620662, -0.1020983
    0.0434763, 0.0845904, -0.0832755, -0.1269837, 0.0828277, 0.0483789, 0.1037824, 0.0571072
    0.0732775, 0.0945174, 0.0561309, 0.0745051, 0.0411969, -0.0275254, -0.0132666, -0.0425338
    -0.1354136, -0.0712286, -0.1289035, -0.0853903, 0.0509822, 0.1508623, 0.0092200, 0.0800618
    0.0208611, -0.0125789, -0.0889751, 0.0254236, -0.1356756, 0.1466179, -0.1343241, -0.0881316
    0.0382349, 0.0085298, 0.1335090, 0.1698340, -0.0733378, 0.1544804, 0.0720860, -0.0480656
    0.0, 0.0, 0.0, 0.0, 0.0, 0.0, 0.0, 0.0
    0.0, 0.0, 0.0, 0.0, 0.0, 0.0, 0.0, 0.0];

   // BsplineLUT 'l1_bspline': grid(15 pts) + table(4×16×15)
   w3 : ARRAY[0..14] OF REAL :=
[-3.0000000, -2.5714286, -2.1428571, -1.7142857, -1.2857143, -0.8571429, -0.4285714, 0.0
    0.4285714, 0.8571429, 1.2857143, 1.7142857, 2.1428571, 2.5714286, 3.0000000];
   w4 : ARRAY[0..959] OF REAL :=
[-0.1185466, -0.1611836, -0.1728346, -0.1652838, -0.1499100, -0.1263157, -0.0918775, -0.0506642
    -0.0106035, 0.0205325, 0.0352327, 0.0306995, 0.0176215, 0.0077084, 0.0028762, 0.1164080
    0.1550023, 0.1593884, 0.1416416, 0.1134742, 0.0746018, 0.0233048, -0.0269650, -0.0544395
    -0.0535770, -0.0395074, -0.0252383, -0.0138686, -0.0064940, -0.0025418, 0.1212922, 0.1619404
    0.1678115, 0.1523909, 0.1282051, 0.0928486, 0.0419677, -0.0115294, -0.0451882, -0.0519172
    -0.0442232, -0.0331994, -0.0222638, -0.0132838, -0.0068407, -0.0936515, -0.1284898, -0.1399855
    -0.1367440, -0.1264903, -0.1057708, -0.0699268, -0.0297622, -0.0046321, -0.0001142, -0.0042117
    -0.0068977, -0.0070424, -0.0052009, -0.0026190, 0.1094929, 0.1466373, 0.1529748, 0.1407870
    0.1210990, 0.0899560, 0.0415844, -0.0111175, -0.0448951, -0.0520181, -0.0445710, -0.0334057
    -0.0221790, -0.0130453, -0.0066071, 0.1187390, 0.1585028, 0.1642579, 0.1493950, 0.1262221
    0.0918142, 0.0412989, -0.0121866, -0.0455425, -0.0516198, -0.0436172, -0.0330280, -0.0226940
    -0.0138372, -0.0071373, 0.0376654, 0.0675727, 0.1009731, 0.1242983, 0.1263663, 0.1084614
    0.0752697, 0.0349018, -0.0026205, -0.0296893, -0.0417853, -0.0377709, -0.0256473, -0.0141969
    -0.0061970, 0.1184750, 0.1574777, 0.1612365, 0.1417943, 0.1112666, 0.0713156, 0.0221729
    -0.0245199, -0.0508939, -0.0522951, -0.0408964, -0.0274740, -0.0156899, -0.0076179, -0.0030719
    0.0231729, 0.0570810, 0.1052454, 0.1414796, 0.1442100, 0.1182180, 0.0748846, 0.0268722
    -0.0125737, -0.0359832, -0.0432108, -0.0365266, -0.0237850, -0.0129781, -0.0060276, 0.0068627
    0.0288937, 0.0653519, 0.0969420, 0.1071390, 0.0971053, 0.0724051, 0.0391903, 0.0039750
    -0.0258812, -0.0419582, -0.0400625, -0.0283319, -0.0162498, -0.0072578, -0.1194447, -0.1587159
    -0.1644049, -0.1540088, -0.1434027, -0.1299989, -0.1072404, -0.0742334, -0.0335070, 0.0067950
    0.0314785, 0.0319794, 0.0200713, 0.0096345, 0.0037933, 0.1133275, 0.1547838, 0.1663608
    0.1563906, 0.1331545, 0.0957848, 0.0427152, -0.0120714, -0.0460413, -0.0522769, -0.0437640
    -0.0320173, -0.0206554, -0.0116729, -0.0055405, 0.0739314, 0.1109307, 0.1370489, 0.1485064
    0.1427782, 0.1199667, 0.0814974, 0.0355972, -0.0056830, -0.0340867, -0.0462228, -0.0418843
    -0.0291076, -0.0166036, -0.0074544, 0.1246268, 0.1663985, 0.1722501, 0.1555205, 0.1291907
    0.0934859, 0.0466661, -0.0012864, -0.0339111, -0.0453605, -0.0433240, -0.0352212, -0.0251985
    -0.0164961, -0.0100727, 0.0280062, 0.0545171, 0.0871669, 0.1114988, 0.1152633, 0.0987976
    0.0660465, 0.0261479, -0.0088806, -0.0313755, -0.0392330, -0.0331661, -0.0209484, -0.0107304
    -0.0044195, -0.0804502, -0.1115401, -0.1237563, -0.1238746, -0.1178652, -0.1022079, -0.0722860
    -0.0358783, -0.0076977, 0.0056848, 0.0081148, 0.0042526, -0.0008231, -0.0026550, -0.0017083
    -0.1075111, -0.1513139, -0.1707310, -0.1697639, -0.1519884, -0.1123527, -0.0463838, 0.0232968
    0.0591967, 0.0520882, 0.0287567, 0.0113045, 0.0017425, -0.0016278, -0.0013955, -0.1163130
    -0.1543022, -0.1551655, -0.1249785, -0.0737230, -0.0174902, 0.0268795, 0.0500879, 0.0474698
    0.0245961, -0.0000769, -0.0126992, -0.0150247, -0.0115051, -0.0059861, -0.1221146, -0.1629714
    -0.1693566, -0.1565035, -0.1384852, -0.1131765, -0.0755465, -0.0313306, 0.0076217, 0.0331493
    0.0418592, 0.0339687, 0.0191801, 0.0077054, 0.0013899, -0.0946115, -0.1247946, -0.1207554
    -0.0790445, -0.0051254, 0.0661646, 0.0963625, 0.0830347, 0.0445621, -0.0001126, -0.0316626
    -0.0382396, -0.0295385, -0.0180286, -0.0086210, -0.1111198, -0.1485720, -0.1550920, -0.1448162
    -0.1307577, -0.1108971, -0.0803174, -0.0420704, -0.0038105, 0.0267422, 0.0418592, 0.0382153
    0.0251295, 0.0131010, 0.0050240, -0.1198157, -0.1598088, -0.1658826, -0.1530319, -0.1350904
    -0.1098848, -0.0724105, -0.0287039, 0.0089435, 0.0325894, 0.0398976, 0.0317844, 0.0174705
    0.0065388, 0.0006581, -0.0224338, -0.0511973, -0.0914252, -0.1246627, -0.1355763, -0.1268838
    -0.1053253, -0.0735197, -0.0319071, 0.0117056, 0.0401575, 0.0430635, 0.0312201, 0.0179805
    0.0080600, -0.1183016, -0.1565961, -0.1564034, -0.1230801, -0.0665991, -0.0058225, 0.0393167
    0.0600484, 0.0542909, 0.0289250, 0.0020724, -0.0126118, -0.0163713, -0.0131443, -0.0071311
    -0.0126077, -0.0451542, -0.0946705, -0.1259195, -0.1110194, -0.0623395, -0.0022841, 0.0452215
    0.0560221, 0.0297608, -0.0037888, -0.0214686, -0.0246745, -0.0191550, -0.0104662, -0.0067350
    -0.0287952, -0.0658434, -0.0997334, -0.1146822, -0.1107441, -0.0917863, -0.0609132, -0.0209531
    0.0192219, 0.0430905, 0.0412662, 0.0262611, 0.0129130, 0.0048849, -0.1192570, -0.1612922
    -0.1718575, -0.1647822, -0.1518551, -0.1260223, -0.0777507, -0.0190807, 0.0258406, 0.0456150
    0.0451751, 0.0315832, 0.0150039, 0.0048415, 0.0012090, -0.1128102, -0.1535935, -0.1583066
    -0.1199614, -0.0414408, 0.0409846, 0.0861816, 0.0865232, 0.0538921, 0.0063032, -0.0307722
    -0.0406204, -0.0330485, -0.0214716, -0.0113644, -0.0630026, -0.0989624, -0.1293125, -0.1462803
    -0.1446681, -0.1291148, -0.1061113, -0.0764903, -0.0380279, 0.0038057, 0.0337559, 0.0418607
    0.0351598, 0.0231704, 0.0114830, -0.1249874, -0.1670758, -0.1743109, -0.1625542, -0.1467603
    -0.1263812, -0.0974452, -0.0598267, -0.0157750, 0.0267821, 0.0527706, 0.0533988, 0.0392336
    0.0231458, 0.0098816, -0.0167747, -0.0431118, -0.0821729, -0.1156180, -0.1276861, -0.1188111
    -0.0935042, -0.0572893, -0.0163505, 0.0203483, 0.0403404, 0.0372682, 0.0229628, 0.0109925
    0.0042679, -0.0816420, -0.1062761, -0.1001644, -0.0616535, 0.0034427, 0.0653489, 0.0913248
    0.0779446, 0.0388183, -0.0083070, -0.0407165, -0.0444709, -0.0317437, -0.0179014, -0.0079489
    0.0151975, 0.0235521, 0.0332792, 0.0507921, 0.0777826, 0.0953368, 0.0822438, 0.0450360
    0.0060403, -0.0205440, -0.0310559, -0.0257163, -0.0139482, -0.0056028, -0.0019484, -0.1155580
    -0.1545806, -0.1588712, -0.1360652, -0.0957358, -0.0456954, 0.0059780, 0.0441973, 0.0503743
    0.0259233, -0.0023669, -0.0144551, -0.0143574, -0.0098370, -0.0048087, -0.1205282, -0.1611996
    -0.1623739, -0.1234019, -0.0511928, 0.0254091, 0.0743054, 0.0848094, 0.0589316, 0.0110262
    -0.0291269, -0.0411464, -0.0344836, -0.0228228, -0.0121515, -0.1043956, -0.1424929, -0.1545623
    -0.1525580, -0.1475409, -0.1377990, -0.1186325, -0.0868331, -0.0403469, 0.0120998, 0.0481567
    0.0537229, 0.0408979, 0.0251194, 0.0123837, -0.1087387, -0.1459541, -0.1485932, -0.1171993
    -0.0579764, 0.0078267, 0.0563506, 0.0746207, 0.0563996, 0.0120958, -0.0269175, -0.0387077
    -0.0323160, -0.0212188, -0.0111836, -0.1180905, -0.1579310, -0.1598222, -0.1251487, -0.0613494
    0.0084301, 0.0585071, 0.0764511, 0.0579023, 0.0139213, -0.0250378, -0.0376370, -0.0322898
    -0.0217316, -0.0117315, -0.0251379, -0.0540239, -0.0928757, -0.1241432, -0.1331588, -0.1218686
    -0.0962172, -0.0613322, -0.0219552, 0.0140414, 0.0348204, 0.0341073, 0.0223325, 0.0116203
    0.0050015, -0.1177874, -0.1573024, -0.1619444, -0.1417454, -0.1074021, -0.0621048, -0.0085318
    0.0372685, 0.0521067, 0.0339863, 0.0078496, -0.0067779, -0.0108954, -0.0090408, -0.0048906
    -0.0120417, -0.0447098, -0.0971188, -0.1399086, -0.1490568, -0.1315648, -0.1013589, -0.0653960
    -0.0266862, 0.0089624, 0.0321423, 0.0373486, 0.0309462, 0.0208850, 0.0113536, -0.0069750
    -0.0289371, -0.0654936, -0.0982360, -0.1114271, -0.1063990, -0.0884556, -0.0606958, -0.0250868
    0.0112298, 0.0345482, 0.0367103, 0.0266989, 0.0155451, 0.0071470, 0.1188454, 0.1575531
    0.1615340, 0.1458852, 0.1252960, 0.1013168, 0.0725062, 0.0397800, 0.0055150, -0.0242361
    -0.0387942, -0.0329794, -0.0182556, -0.0075002, -0.0025888, -0.1122213, -0.1540768, -0.1676361
    -0.1619918, -0.1458810, -0.1176921, -0.0745038, -0.0257562, 0.0122202, 0.0321316, 0.0382330
    0.0353320, 0.0276915, 0.0191909, 0.0116818, -0.0633601, -0.0993192, -0.1294454, -0.1460750
    -0.1434730, -0.1231374, -0.0887078, -0.0474956, -0.0088845, 0.0194919, 0.0322518, 0.0279761
    0.0162082, 0.0072343, 0.0027652, -0.1238974, -0.1653246, -0.1640291, -0.1149265, -0.0239744
    0.0664812, 0.1093154, 0.0991432, 0.0547696, -0.0015556, -0.0436018, -0.0546247, -0.0458544
    -0.0322604, -0.0199737, -0.0225191, -0.0490759, -0.0853007, -0.1152470, -0.1253413, -0.1162182
    -0.0920650, -0.0577134, -0.0184517, 0.0173353, 0.0373541, 0.0351925, 0.0220467, 0.0108314
    0.0044042, -0.0905067, -0.1246435, -0.1371959, -0.1375610, -0.1345223, -0.1268024, -0.1106224
    -0.0818949, -0.0366904, 0.0165826, 0.0539035, 0.0597753, 0.0460540, 0.0282559, 0.0132754
    0.1027418, 0.1458940, 0.1662828, 0.1649976, 0.1437322, 0.1007277, 0.0354482, -0.0318456
    -0.0695069, -0.0686447, -0.0493544, -0.0292685, -0.0135997, -0.0047961, -0.0014169, -0.1171014
    -0.1556434, -0.1607976, -0.1483480, -0.1335257, -0.1178635, -0.0993047, -0.0735262, -0.0352015
    0.0098080, 0.0414661, 0.0468319, 0.0359529, 0.0219121, 0.0102643, -0.1203817, -0.1605767
    -0.1667812, -0.1542558, -0.1381546, -0.1216702, -0.1045547, -0.0815037, -0.0446325, 0.0014981
    0.0365366, 0.0467486, 0.0403142, 0.0285137, 0.0169089, 0.1002332, 0.1354359, 0.1425826
    0.1294305, 0.1047949, 0.0734366, 0.0392145, 0.0069307, -0.0181247, -0.0327154, -0.0362152
    -0.0297695, -0.0191288, -0.0102292, -0.0045105, -0.1082906, -0.1448953, -0.1514328, -0.1415441
    -0.1285956, -0.1145728, -0.0983684, -0.0758803, -0.0415573, -0.0001217, 0.0306798, 0.0390608
    0.0327519, 0.0221901, 0.0123327, -0.1177685, -0.1570408, -0.1630592, -0.1509109, -0.1355683
    -0.1202167, -0.1046190, -0.0832344, -0.0477946, -0.0023018, 0.0336691, 0.0464788, 0.0424047
    0.0308316, 0.0179980, -0.0274415, -0.0552075, -0.0829036, -0.0743872, -0.0079748, 0.0719735
    0.1095986, 0.0964300, 0.0514424, -0.0031709, -0.0415716, -0.0478322, -0.0351535, -0.0203725
    -0.0092955, -0.1190558, -0.1580338, -0.1628482, -0.1496336, -0.1340558, -0.1181711, -0.1003914
    -0.0760892, -0.0391883, 0.0051607, 0.0375761, 0.0452217, 0.0366817, 0.0235403, 0.0115771
    -0.0122453, -0.0452500, -0.0982542, -0.1418979, -0.1524913, -0.1386983, -0.1158748, -0.0867925
    -0.0472319, -0.0030324, 0.0271305, 0.0316634, 0.0216764, 0.0109768, 0.0038074, 0.0056665
    0.0203240, 0.0455025, 0.0729728, 0.0945766, 0.1057540, 0.1027918, 0.0816016, 0.0382571
    -0.0172831, -0.0574904, -0.0642684, -0.0498448, -0.0306137, -0.0141799, -0.1132877, -0.1423928
    -0.1257204, -0.0690783, 0.0124324, 0.0772630, 0.0827558, 0.0403378, -0.0078174, -0.0370361
    -0.0452796, -0.0351606, -0.0184718, -0.0071259, -0.0023027, -0.1139212, -0.1553163, -0.1672838
    -0.1607169, -0.1467058, -0.1274866, -0.1029656, -0.0714867, -0.0307369, 0.0125788, 0.0403341
    0.0416061, 0.0282631, 0.0148155, 0.0057112, -0.0609488, -0.0963577, -0.1260219, -0.1395709
    -0.1284558, -0.0917699, -0.0326726, 0.0236884, 0.0403581, 0.0129372, -0.0215786, -0.0349511
    -0.0317258, -0.0217525, -0.0110394, -0.1244168, -0.1660250, -0.1723339, -0.1584518, -0.1393272
    -0.1175164, -0.0925129, -0.0636112, -0.0301276, 0.0035928, 0.0268426, 0.0329896, 0.0282779
    0.0206643, 0.0139797, -0.0124840, -0.0339846, -0.0592003, -0.0530296, 0.0060139, 0.0761174
    0.1045475, 0.0849964, 0.0380051, -0.0141146, -0.0472311, -0.0474186, -0.0303917, -0.0151116
    -0.0061100, 0.0868751, 0.1178409, 0.1253527, 0.1169635, 0.1003876, 0.0767242, 0.0459131
    0.0125569, -0.0161009, -0.0347057, -0.0403378, -0.0329215, -0.0200967, -0.0099572, -0.0040698];

   // MatMul 'l1_base': W(4×16) + b(4)
   w5 : ARRAY[0..67] OF REAL :=
[0.0227410, -0.0533916, -0.0561938, -0.0049936, -0.0590683, -0.0565307, -0.0560681, -0.0494344
    -0.0503630, -0.0591014, 0.0313365, -0.0618064, -0.0624162, -0.0619019, -0.0512237, 0.0036076
    0.0312500, -0.0205478, 0.0405237, -0.0518004, 0.0497862, 0.0367622, 0.0530868, -0.0234220
    -0.0351746, 0.0666708, 0.0426824, -0.0580829, 0.0508394, 0.0829995, 0.0470647, -0.0636629
    -0.0366331, -0.0168737, -0.0585914, 0.0710758, -0.0545160, -0.0535938, 0.0407549, -0.0097806
    0.0396265, 0.0398606, -0.0378223, 0.0598480, 0.0338706, -0.0801397, 0.0446221, 0.0936506
    -0.0425605, 0.0566664, 0.0594682, -0.0393109, 0.0490207, 0.0593235, -0.0528647, 0.0505356
    0.0425443, -0.0891089, -0.0422298, 0.0501610, -0.0416037, 0.0420642, -0.0542606, -0.0447944
    0.0, 0.0, 0.0, 0.0];

   // Total: 6 array blocks
   END_STRUCT;
BEGIN
END_DATA_BLOCK

FUNCTION "BsplineEval" : REAL
{ S7_Optimized_Access := 'FALSE' }
VERSION : 0.1
VAR_INPUT
    x : REAL;
    lut_grid : ARRAY[0..14] OF REAL;
    lut_table : ARRAY[0..14] OF REAL;
END_VAR
VAR_TEMP
    lo, hi, mid : INT;
    t, vlo, vhi : REAL;
END_VAR

BEGIN
    // Binary search for interval containing x
    lo := 0;
    hi := 14;
    WHILE hi - lo > 1 DO
        mid := lo + (hi - lo) / 2;
        IF x > lut_grid[mid] THEN lo := mid; ELSE hi := mid; END_IF;
    END_WHILE;

    // Linear interpolation: y = vlo*(1-t) + vhi*t
    vlo := lut_table[lo];
    vhi := lut_table[hi];
    t := (x - lut_grid[lo]) / (lut_grid[hi] - lut_grid[lo] + 1.0E-10);
    "BsplineEval" := vlo * (1.0 - t) + vhi * t;
END_FUNCTION

FUNCTION_BLOCK "NeuroPLC_Inference"
{ S7_Optimized_Access := 'FALSE' }
VERSION : 0.1
VAR_INPUT
    features : ARRAY[0..27] OF REAL;
END_VAR

VAR_OUTPUT
    fault_class : INT;
    confidence : REAL;
END_VAR

VAR
    i, j, k : INT;
    sum_val, max_val, t_val : REAL;
    v0 : ARRAY[0..27] OF REAL;
    v1 : ARRAY[0..27] OF REAL;
    v3 : ARRAY[0..15, 0..27] OF REAL;
    v2 : ARRAY[0..15] OF REAL;
    v4 : ARRAY[0..15] OF REAL;
    v5 : ARRAY[0..15] OF REAL;
    v7 : ARRAY[0..3, 0..15] OF REAL;
    v6 : ARRAY[0..3] OF REAL;
    v8 : ARRAY[0..3] OF REAL;
    v9 : ARRAY[0..3] OF REAL;
    lut_tmp : ARRAY[0..14] OF REAL;
END_VAR

BEGIN
    // ---- Input ----
    FOR i := 0 TO 27 DO
        v0[i] := features[i];
    END_FOR;

